C01819=1068.926,-95.070,-58.479,172.290,23.008,154.216
C01820=1068.921,-95.321,-58.468,172.288,23.007,154.216
C01821=1068.914,-95.570,-58.458,172.287,23.005,154.216
C01822=1068.909,-95.820,-58.448,172.285,23.004,154.216
C01823=1068.902,-96.069,-58.438,172.284,23.003,154.216
C01824=1068.897,-96.318,-58.427,172.282,23.001,154.216
C01825=1068.890,-96.568,-58.417,172.280,23.000,154.216
C01826=1068.884,-96.818,-58.406,172.279,22.999,154.216
C01827=1068.878,-97.068,-58.396,172.277,22.997,154.216
C01828=1068.872,-97.318,-58.386,172.275,22.996,154.216
C01829=1068.866,-97.568,-58.376,172.274,22.995,154.216
C01830=1068.859,-97.850,-58.365,172.272,22.993,154.215
C01831=1068.852,-98.133,-58.353,172.270,22.991,154.215
C01832=1068.845,-98.416,-58.341,172.268,22.990,154.215
C01833=1068.838,-98.698,-58.330,172.267,22.989,154.215
C01834=1068.833,-98.948,-58.319,172.265,22.987,154.215
C01835=1068.827,-99.197,-58.309,172.263,22.986,154.215
C01836=1068.820,-99.447,-58.299,172.261,22.985,154.215
C01837=1068.814,-99.697,-58.289,172.260,22.984,154.215
C01838=1068.808,-99.947,-58.278,172.258,22.982,154.215
C01839=1068.801,-100.196,-58.269,172.257,22.981,154.215
C01840=1068.796,-100.446,-58.258,172.255,22.980,154.215
C01841=1068.789,-100.696,-58.248,172.253,22.978,154.215
C01842=1068.783,-100.945,-58.239,172.252,22.977,154.215
C01843=1068.777,-101.195,-58.229,172.250,22.976,154.215
C01844=1068.771,-101.445,-58.218,172.248,22.975,154.215
C01845=1068.764,-101.695,-58.208,172.247,22.974,154.215
C01846=1068.758,-101.944,-58.198,172.245,22.972,154.215
C01847=1068.753,-102.194,-58.188,172.243,22.971,154.215
C01848=1068.746,-102.444,-58.178,172.242,22.970,154.215
C01849=1068.740,-102.693,-58.168,172.240,22.968,154.215
C01850=1068.734,-102.943,-58.157,172.238,22.968,154.216
C01851=1068.728,-103.193,-58.148,172.237,22.966,154.215
C01852=1068.722,-103.443,-58.138,172.235,22.965,154.215
C01853=1068.716,-103.692,-58.127,172.234,22.964,154.215
C01854=1068.710,-103.942,-58.118,172.232,22.962,154.215
C01855=1068.704,-104.192,-58.108,172.230,22.961,154.215
C01856=1068.697,-104.441,-58.098,172.228,22.960,154.216
C01857=1068.692,-104.691,-58.088,172.227,22.959,154.216
C01858=1068.686,-104.941,-58.078,172.225,22.958,154.216
C01859=1068.680,-105.191,-58.069,172.224,22.956,154.216
C01860=1068.673,-105.440,-58.058,172.222,22.956,154.216
C01861=1068.667,-105.691,-58.048,172.220,22.954,154.216
C01862=1068.661,-105.940,-58.038,172.219,22.953,154.216
C01863=1068.654,-106.189,-58.028,172.217,22.952,154.216
C01864=1068.648,-106.439,-58.018,172.215,22.951,154.216
C01865=1068.643,-106.689,-58.008,172.213,22.949,154.216
C01866=1068.637,-106.939,-57.999,172.212,22.948,154.216
C01867=1068.630,-107.188,-57.988,172.210,22.947,154.216
C01868=1068.624,-107.438,-57.979,172.208,22.946,154.216
C01869=1068.618,-107.688,-57.969,172.207,22.945,154.216
C01870=1068.612,-107.938,-57.959,172.205,22.943,154.216
C01871=1068.606,-108.188,-57.949,172.203,22.943,154.216
C01872=1068.600,-108.437,-57.939,172.202,22.941,154.216
C01873=1068.594,-108.687,-57.930,172.200,22.940,154.216
C01874=1068.587,-108.937,-57.920,172.198,22.939,154.216
C01875=1068.581,-109.186,-57.910,172.197,22.938,154.216
C01876=1068.575,-109.436,-57.901,172.195,22.937,154.216
C01877=1068.569,-109.685,-57.891,172.193,22.936,154.216
C01878=1068.562,-109.935,-57.881,172.191,22.935,154.216
C01879=1068.557,-110.185,-57.871,172.190,22.934,154.216
C01880=1068.551,-110.435,-57.861,172.188,22.932,154.216
C01881=1068.545,-110.685,-57.852,172.187,22.932,154.216
C01882=1068.539,-110.935,-57.842,172.186,22.931,154.216
C01883=1068.532,-111.185,-57.833,172.184,22.930,154.216
C01884=1068.526,-111.434,-57.822,172.182,22.929,154.216
C01885=1068.520,-111.683,-57.813,172.181,22.928,154.216
C01886=1068.514,-111.933,-57.803,172.179,22.926,154.216
C01887=1068.507,-112.183,-57.794,172.177,22.925,154.216
C01888=1068.501,-112.433,-57.784,172.175,22.924,154.216
C01889=1068.495,-112.683,-57.774,172.174,22.923,154.216
C01890=1068.490,-112.933,-57.764,172.172,22.922,154.217
C01891=1068.483,-113.183,-57.755,172.170,22.921,154.217
C01892=1068.478,-113.432,-57.746,172.169,22.920,154.217
C01893=1068.472,-113.681,-57.736,172.167,22.919,154.217
C01894=1068.465,-113.962,-57.725,172.165,22.918,154.217
C01895=1068.458,-114.243,-57.714,172.163,22.916,154.217
C01896=1068.450,-114.522,-57.704,172.161,22.916,154.217
C01897=1068.443,-114.803,-57.693,172.159,22.914,154.217
C01898=1068.437,-115.053,-57.683,172.157,22.913,154.217
C01899=1068.431,-115.303,-57.674,172.156,22.912,154.217
C01900=1068.425,-115.552,-57.664,172.154,22.911,154.217
C01901=1068.419,-115.802,-57.654,172.152,22.910,154.217
C01902=1068.413,-116.052,-57.645,172.151,22.909,154.217
C01903=1068.406,-116.302,-57.635,172.149,22.909,154.217
C01904=1068.400,-116.552,-57.626,172.147,22.907,154.217
C01905=1068.395,-116.801,-57.616,172.145,22.906,154.217
C01906=1068.389,-117.050,-57.607,172.144,22.906,154.218
C01907=1068.382,-117.300,-57.597,172.143,22.905,154.217
C01908=1068.376,-117.550,-57.588,172.141,22.904,154.218
C01909=1068.370,-117.800,-57.578,172.139,22.903,154.218
C01910=1068.364,-118.050,-57.569,172.138,22.902,154.218
C01911=1068.358,-118.300,-57.560,172.136,22.901,154.218
C01912=1068.351,-118.550,-57.551,172.134,22.900,154.218
C01913=1068.345,-118.799,-57.541,172.132,22.899,154.218
C01914=1068.339,-119.049,-57.532,172.131,22.898,154.218
C01915=1068.333,-119.298,-57.522,172.129,22.897,154.218
C01916=1068.327,-119.548,-57.513,172.127,22.896,154.218
C01917=1068.321,-119.798,-57.503,172.125,22.895,154.218
C01918=1068.315,-120.048,-57.494,172.124,22.895,154.218
C01919=1068.308,-120.297,-57.484,172.122,22.893,154.218
C01920=1068.303,-120.548,-57.475,172.120,22.893,154.218
C01921=1068.296,-120.798,-57.466,172.118,22.892,154.219
C01922=1068.289,-121.047,-57.457,172.117,22.890,154.219
C01923=1068.284,-121.296,-57.448,172.115,22.890,154.219
C01924=1068.278,-121.546,-57.438,172.113,22.889,154.219
C01925=1068.272,-121.796,-57.428,172.111,22.888,154.219
C01926=1068.265,-122.046,-57.419,172.110,22.887,154.219
C01927=1068.260,-122.296,-57.410,172.109,22.886,154.219
C01928=1068.253,-122.546,-57.401,172.107,22.886,154.219
C01929=1068.247,-122.795,-57.392,172.105,22.885,154.219
C01930=1068.241,-123.044,-57.382,172.103,22.884,154.219
C01931=1068.235,-123.294,-57.373,172.102,22.883,154.219
C01932=1068.229,-123.545,-57.364,172.100,22.882,154.219
C01933=1068.223,-123.794,-57.354,172.098,22.881,154.219
C01934=1068.217,-124.044,-57.345,172.096,22.880,154.220
C01935=1068.210,-124.293,-57.336,172.095,22.880,154.220
C01936=1068.204,-124.543,-57.327,172.093,22.879,154.220
C01937=1068.198,-124.793,-57.318,172.091,22.878,154.220
C01938=1068.192,-125.043,-57.308,172.089,22.877,154.220
C01939=1068.185,-125.292,-57.299,172.088,22.876,154.220
C01940=1068.180,-125.542,-57.291,172.086,22.875,154.220
C01941=1068.174,-125.792,-57.281,172.084,22.875,154.220
C01942=1068.167,-126.042,-57.272,172.083,22.874,154.220
C01943=1068.161,-126.291,-57.263,172.081,22.873,154.220
C01944=1068.155,-126.542,-57.254,172.079,22.873,154.221
C01945=1068.149,-126.791,-57.244,172.078,22.872,154.221
C01946=1068.142,-127.040,-57.236,172.076,22.871,154.221
C01947=1068.136,-127.291,-57.227,172.074,22.870,154.221
C01948=1068.130,-127.540,-57.217,172.072,22.870,154.221
C01949=1068.124,-127.790,-57.208,172.070,22.869,154.221
C01950=1068.118,-128.041,-57.199,172.069,22.868,154.221
C01951=1068.115,-128.291,-57.188,172.067,22.866,154.221
C01952=1068.113,-128.542,-57.178,172.066,22.863,154.221
C01953=1068.113,-128.793,-57.166,172.065,22.860,154.220
C01954=1068.115,-129.046,-57.153,172.064,22.856,154.220
C01955=1068.119,-129.298,-57.140,172.064,22.852,154.219
C01956=1068.125,-129.549,-57.125,172.064,22.847,154.218
C01957=1068.132,-129.799,-57.110,172.064,22.841,154.217
C01958=1067.743,-129.822,-57.282,172.016,22.987,154.250
C01959=1067.737,-129.572,-57.297,172.017,22.993,154.251
C01960=1067.732,-129.320,-57.312,172.017,22.997,154.252
C01961=1067.727,-129.068,-57.325,172.018,23.002,154.252
C01962=1067.725,-128.816,-57.338,172.018,23.005,154.253
C01963=1067.725,-128.565,-57.350,172.019,23.009,154.254
C01964=1067.726,-128.314,-57.361,172.020,23.011,154.254
C01965=1067.730,-128.063,-57.371,172.021,23.013,154.254
C01966=1067.736,-127.812,-57.381,172.023,23.014,154.254
C01967=1067.742,-127.563,-57.390,172.025,23.015,154.254
C01968=1067.747,-127.313,-57.399,172.027,23.015,154.254
C01969=1067.754,-127.063,-57.408,172.029,23.016,154.254
C01970=1067.760,-126.814,-57.417,172.030,23.017,154.253
C01971=1067.766,-126.564,-57.427,172.032,23.018,154.253
C01972=1067.773,-126.314,-57.436,172.034,23.018,154.253
C01973=1067.778,-126.065,-57.444,172.036,23.019,154.253
C01974=1067.785,-125.815,-57.454,172.037,23.021,154.253
C01975=1067.791,-125.565,-57.463,172.039,23.021,154.253
C01976=1067.797,-125.315,-57.472,172.040,23.022,154.253
C01977=1067.804,-125.065,-57.481,172.042,23.022,154.253
C01978=1067.810,-124.815,-57.491,172.044,23.023,154.253
C01979=1067.815,-124.566,-57.500,172.045,23.024,154.253
C01980=1067.822,-124.316,-57.508,172.047,23.025,154.252
C01981=1067.828,-124.066,-57.518,172.049,23.025,154.252
C01982=1067.834,-123.816,-57.527,172.051,23.027,154.252
C01983=1067.840,-123.567,-57.537,172.053,23.028,154.252
C01984=1067.846,-123.317,-57.545,172.054,23.028,154.252
C01985=1067.852,-123.067,-57.555,172.056,23.029,154.252
C01986=1067.859,-122.818,-57.564,172.058,23.030,154.252
C01987=1067.865,-122.568,-57.573,172.060,23.031,154.252
C01988=1067.871,-122.318,-57.583,172.061,23.032,154.252
C01989=1067.877,-122.068,-57.593,172.063,23.033,154.252
C01990=1067.883,-121.819,-57.601,172.065,23.033,154.252
C01991=1067.889,-121.569,-57.611,172.067,23.034,154.251
C01992=1067.896,-121.319,-57.620,172.068,23.035,154.251
C01993=1067.902,-121.069,-57.629,172.070,23.036,154.251
C01994=1067.908,-120.820,-57.639,172.071,23.037,154.251
C01995=1067.914,-120.570,-57.648,172.073,23.038,154.251
C01996=1067.920,-120.319,-57.657,172.075,23.039,154.251
C01997=1067.926,-120.070,-57.666,172.076,23.039,154.251
C01998=1067.932,-119.821,-57.676,172.078,23.040,154.251
C01999=1067.938,-119.571,-57.685,172.080,23.042,154.251
C02000=1067.944,-119.321,-57.695,172.082,23.042,154.251
C02001=1067.951,-119.071,-57.704,172.083,23.043,154.251
C02002=1067.957,-118.822,-57.714,172.085,23.044,154.251
C02003=1067.963,-118.572,-57.723,172.087,23.045,154.251
C02004=1067.970,-118.322,-57.733,172.089,23.046,154.251
C02005=1067.976,-118.072,-57.742,172.090,23.047,154.251
C02006=1067.981,-117.823,-57.751,172.092,23.048,154.250
C02007=1067.987,-117.573,-57.760,172.094,23.049,154.250
C02008=1067.993,-117.323,-57.770,172.095,23.050,154.250
C02009=1067.999,-117.073,-57.779,172.097,23.051,154.250
C02010=1068.006,-116.823,-57.789,172.099,23.052,154.250
C02011=1068.012,-116.574,-57.799,172.101,23.053,154.250
C02012=1068.018,-116.324,-57.808,172.103,23.054,154.250
C02013=1068.024,-116.074,-57.818,172.104,23.055,154.250
C02014=1068.030,-115.824,-57.827,172.106,23.056,154.250
C02015=1068.037,-115.574,-57.837,172.108,23.056,154.250
C02016=1068.043,-115.325,-57.846,172.109,23.058,154.250
C02017=1068.049,-115.075,-57.856,172.110,23.058,154.250
C02018=1068.054,-114.826,-57.865,172.112,23.059,154.250
C02019=1068.062,-114.545,-57.876,172.115,23.061,154.250
C02020=1068.069,-114.265,-57.887,172.116,23.062,154.250
C02021=1068.076,-113.984,-57.898,172.118,23.063,154.249
C02022=1068.083,-113.703,-57.908,172.120,23.064,154.250
C02023=1068.089,-113.453,-57.918,172.122,23.065,154.249
C02024=1068.095,-113.205,-57.928,172.123,23.066,154.249
C02025=1068.101,-112.955,-57.937,172.125,23.067,154.249
C02026=1068.107,-112.705,-57.947,172.127,23.068,154.249
C02027=1068.113,-112.455,-57.957,172.128,23.069,154.249
C02028=1068.119,-112.205,-57.967,172.130,23.070,154.249
C02029=1068.125,-111.955,-57.976,172.132,23.072,154.249
C02030=1068.131,-111.706,-57.986,172.133,23.072,154.249
C02031=1068.137,-111.456,-57.995,172.135,23.074,154.249
C02032=1068.144,-111.206,-58.005,172.137,23.074,154.249
C02033=1068.150,-110.956,-58.014,172.139,23.076,154.249
C02034=1068.156,-110.707,-58.025,172.140,23.076,154.249
C02035=1068.162,-110.457,-58.034,172.142,23.078,154.249
C02036=1068.169,-110.207,-58.044,172.144,23.079,154.249
C02037=1068.175,-109.958,-58.053,172.145,23.080,154.249
C02038=1068.180,-109.707,-58.063,172.147,23.081,154.249
C02039=1068.186,-109.458,-58.073,172.149,23.082,154.249
C02040=1068.193,-109.208,-58.083,172.150,23.083,154.249
C02041=1068.199,-108.959,-58.093,172.152,23.085,154.249
C02042=1068.205,-108.709,-58.102,172.154,23.085,154.249
C02043=1068.211,-108.459,-58.112,172.155,23.087,154.249
C02044=1068.218,-108.209,-58.122,172.157,23.087,154.249
C02045=1068.224,-107.960,-58.132,172.159,23.089,154.249
C02046=1068.229,-107.710,-58.142,172.161,23.090,154.249
C02047=1068.236,-107.460,-58.152,172.162,23.091,154.248
C02048=1068.242,-107.210,-58.161,172.164,23.092,154.248
C02049=1068.248,-106.961,-58.171,172.166,23.093,154.248
C02050=1068.254,-106.711,-58.181,172.167,23.094,154.248
C02051=1068.260,-106.461,-58.191,172.169,23.096,154.248
C02052=1068.266,-106.212,-58.201,172.171,23.097,154.248
C02053=1068.273,-105.962,-58.211,172.172,23.098,154.248
C02054=1068.279,-105.713,-58.221,172.174,23.099,154.248
C02055=1068.285,-105.462,-58.231,172.176,23.100,154.248
C02056=1068.291,-105.212,-58.241,172.177,23.102,154.248
C02057=1068.297,-104.963,-58.251,172.179,23.103,154.248
C02058=1068.304,-104.713,-58.261,172.181,23.104,154.248
C02059=1068.309,-104.463,-58.271,172.182,23.105,154.248
C02060=1068.315,-104.214,-58.281,172.184,23.106,154.248
C02061=1068.322,-103.964,-58.291,172.185,23.107,154.248
C02062=1068.328,-103.714,-58.300,172.186,23.109,154.248
C02063=1068.334,-103.465,-58.311,172.188,23.109,154.248
C02064=1068.340,-103.215,-58.321,172.190,23.111,154.248
C02065=1068.346,-102.965,-58.330,172.192,23.112,154.248
C02066=1068.352,-102.715,-58.341,172.193,23.113,154.248
C02067=1068.358,-102.466,-58.351,172.195,23.115,154.248
C02068=1068.364,-102.216,-58.360,172.196,23.116,154.248
C02069=1068.370,-101.967,-58.370,172.198,23.117,154.248
C02070=1068.376,-101.717,-58.381,172.200,23.118,154.248
C02071=1068.383,-101.467,-58.391,172.201,23.119,154.248
C02072=1068.389,-101.217,-58.401,172.203,23.121,154.248
C02073=1068.395,-100.967,-58.411,172.205,23.122,154.248
C02074=1068.401,-100.718,-58.421,172.206,23.123,154.248
C02075=1068.407,-100.468,-58.431,172.208,23.125,154.248
C02076=1068.413,-100.218,-58.442,172.210,23.126,154.248
C02077=1068.419,-99.969,-58.451,172.211,23.127,154.248
C02078=1068.426,-99.719,-58.462,172.213,23.128,154.248
C02079=1068.432,-99.469,-58.472,172.215,23.129,154.248
C02080=1068.438,-99.219,-58.482,172.216,23.131,154.248
C02081=1068.444,-98.970,-58.492,172.218,23.132,154.248
C02082=1068.450,-98.719,-58.502,172.220,23.133,154.248
C02083=1068.457,-98.436,-58.514,172.222,23.135,154.248
C02084=1068.464,-98.154,-58.525,172.224,23.136,154.248
C02085=1068.471,-97.871,-58.537,172.225,23.138,154.248
C02086=1068.477,-97.589,-58.548,172.227,23.139,154.248
C02087=1068.484,-97.339,-58.559,172.230,23.141,154.248
C02088=1068.490,-97.089,-58.569,172.231,23.142,154.248
C02089=1068.496,-96.840,-58.579,172.233,23.143,154.248
C02090=1068.502,-96.590,-58.590,172.234,23.145,154.248
C02091=1068.508,-96.341,-58.600,172.236,23.147,154.248
C02092=1068.514,-96.091,-58.611,172.238,23.148,154.248
C02093=1068.520,-95.841,-58.620,172.239,23.149,154.248
C02094=1068.526,-95.592,-58.631,172.241,23.150,154.248
C02095=1068.532,-95.341,-58.641,172.242,23.152,154.248
C02096=1068.538,-95.092,-58.652,172.244,23.153,154.249
C02097=1068.544,-94.842,-58.663,172.246,23.154,154.249
C02098=1068.550,-94.592,-58.672,172.247,23.156,154.249
C02099=1068.556,-94.343,-58.683,172.249,23.157,154.249
C02100=1068.562,-94.093,-58.693,172.250,23.159,154.249
C02101=1068.568,-93.844,-58.704,172.252,23.160,154.249
C02102=1068.575,-93.594,-58.714,172.254,23.162,154.249
C02103=1068.580,-93.344,-58.724,172.255,23.163,154.249
C02104=1068.586,-93.094,-58.735,172.257,23.164,154.249
C02105=1068.592,-92.844,-58.745,172.259,23.166,154.249
C02106=1068.598,-92.595,-58.756,172.260,23.167,154.249
C02107=1068.605,-92.345,-58.766,172.262,23.169,154.249
C02108=1068.611,-92.095,-58.776,172.263,23.170,154.249
C02109=1068.616,-91.845,-58.787,172.265,23.171,154.249
C02110=1068.623,-91.596,-58.798,172.267,23.173,154.249
C02111=1068.629,-91.347,-58.809,172.268,23.174,154.249
C02112=1068.635,-91.096,-58.818,172.270,23.176,154.249
C02113=1068.641,-90.847,-58.829,172.271,23.177,154.249
C02114=1068.647,-90.597,-58.840,172.273,23.179,154.249
C02115=1068.653,-90.347,-58.850,172.275,23.180,154.249
C02116=1068.659,-90.098,-58.861,172.276,23.181,154.249
C02117=1068.666,-89.848,-58.871,172.278,23.183,154.249
C02118=1068.671,-89.599,-58.882,172.279,23.184,154.249
C02119=1068.677,-89.349,-58.892,172.281,23.186,154.249
C02120=1068.683,-89.099,-58.903,172.283,23.187,154.249
C02121=1068.690,-88.849,-58.914,172.284,23.189,154.250
C02122=1068.696,-88.600,-58.924,172.286,23.190,154.250
C02123=1068.702,-88.350,-58.934,172.287,23.192,154.250
C02124=1068.707,-88.100,-58.945,172.289,23.193,154.250
C02125=1068.714,-87.850,-58.956,172.290,23.195,154.250
C02126=1068.720,-87.601,-58.967,172.292,23.196,154.250
C02127=1068.726,-87.352,-58.978,172.294,23.197,154.250
C02128=1068.733,-87.101,-58.988,172.295,23.199,154.250
C02129=1068.738,-86.852,-58.998,172.297,23.201,154.250
C02130=1068.744,-86.602,-59.009,172.298,23.202,154.250
C02131=1068.751,-86.353,-59.020,172.300,23.203,154.250
C02132=1068.757,-86.103,-59.031,172.301,23.205,154.250
C02133=1068.762,-85.853,-59.041,172.303,23.206,154.250
C02134=1068.769,-85.603,-59.051,172.305,23.208,154.250
C02135=1068.775,-85.353,-59.062,172.306,23.209,154.250
C02136=1068.781,-85.104,-59.073,172.308,23.211,154.250
C02137=1068.787,-84.855,-59.084,172.309,23.212,154.250
C02138=1068.794,-84.604,-59.095,172.311,23.214,154.250
C02139=1068.800,-84.355,-59.106,172.313,23.215,154.250
C02140=1068.806,-84.106,-59.116,172.314,23.217,154.250
C02141=1068.812,-83.855,-59.127,172.316,23.218,154.251
C02142=1068.818,-83.605,-59.137,172.317,23.220,154.251
C02143=1068.824,-83.356,-59.148,172.320,23.222,154.251
C02144=1068.831,-83.106,-59.159,172.321,23.223,154.251
C02145=1068.836,-82.856,-59.170,172.323,23.225,154.251
C02146=1068.843,-82.607,-59.180,172.325,23.226,154.251
C02147=1068.850,-82.326,-59.193,172.326,23.228,154.251
C02148=1068.857,-82.046,-59.205,172.328,23.229,154.251
C02149=1068.864,-81.766,-59.217,172.329,23.231,154.251
C02150=1068.871,-81.486,-59.229,172.332,23.233,154.251
C02151=1068.877,-81.235,-59.241,172.333,23.235,154.251
C02152=1068.883,-80.986,-59.251,172.335,23.236,154.251
C02153=1068.889,-80.737,-59.262,172.336,23.238,154.251
C02154=1068.895,-80.487,-59.273,172.338,23.239,154.251
C02155=1068.902,-80.237,-59.283,172.339,23.241,154.251
C02156=1068.908,-79.987,-59.295,172.341,23.243,154.252
C02157=1068.914,-79.738,-59.306,172.343,23.244,154.252
C02158=1068.920,-79.488,-59.316,172.344,23.246,154.252
C02159=1068.926,-79.238,-59.328,172.346,23.247,154.252
C02160=1068.932,-78.989,-59.339,172.347,23.249,154.252
C02161=1068.938,-78.739,-59.349,172.349,23.250,154.252
C02162=1068.945,-78.489,-59.360,172.350,23.252,154.252
C02163=1068.950,-78.240,-59.371,172.352,23.254,154.252
C02164=1068.957,-77.990,-59.382,172.353,23.255,154.252
C02165=1068.962,-77.740,-59.393,172.355,23.257,154.252
C02166=1068.968,-77.491,-59.404,172.356,23.259,154.252
C02167=1068.975,-77.240,-59.415,172.358,23.260,154.253
C02168=1068.980,-76.991,-59.426,172.360,23.262,154.253
C02169=1068.986,-76.741,-59.437,172.361,23.264,154.253
C02170=1068.993,-76.492,-59.449,172.363,23.266,154.253
C02171=1068.998,-76.242,-59.460,172.365,23.267,154.253
C02172=1069.005,-75.992,-59.471,172.366,23.269,154.253
C02173=1069.010,-75.743,-59.482,172.368,23.270,154.253
C02174=1069.017,-75.492,-59.493,172.370,23.272,154.253
C02175=1069.023,-75.243,-59.503,172.371,23.274,154.253
C02176=1069.029,-74.994,-59.514,172.373,23.275,154.253
C02177=1069.036,-74.744,-59.526,172.374,23.277,154.253
C02178=1069.041,-74.495,-59.537,172.376,23.279,154.253
C02179=1069.048,-74.245,-59.548,172.377,23.281,154.254
C02180=1069.054,-73.995,-59.559,172.379,23.282,154.254
C02181=1069.060,-73.745,-59.570,172.380,23.284,154.254
C02182=1069.066,-73.496,-59.582,172.382,23.286,154.254
C02183=1069.071,-73.246,-59.594,172.383,23.287,154.254
C02184=1069.077,-72.996,-59.605,172.385,23.289,154.254
C02185=1069.083,-72.747,-59.616,172.386,23.291,154.254
C02186=1069.089,-72.496,-59.627,172.388,23.293,154.254
C02187=1069.095,-72.247,-59.638,172.389,23.294,154.254
C02188=1069.101,-71.998,-59.649,172.391,23.296,154.255
C02189=1069.107,-71.747,-59.661,172.392,23.298,154.255
C02190=1069.112,-71.498,-59.672,172.394,23.299,154.255
C02191=1069.119,-71.248,-59.684,172.395,23.301,154.255
C02192=1069.125,-70.999,-59.695,172.397,23.303,154.255
C02193=1069.131,-70.749,-59.706,172.399,23.305,154.255
C02194=1069.137,-70.500,-59.718,172.401,23.307,154.255
C02195=1069.142,-70.250,-59.729,172.402,23.309,154.255
C02196=1069.149,-70.000,-59.740,172.404,23.311,154.255
C02197=1069.155,-69.751,-59.752,172.405,23.312,154.256
C02198=1069.161,-69.501,-59.763,172.407,23.314,154.256
C02199=1069.167,-69.251,-59.774,172.408,23.316,154.256
C02200=1069.173,-69.002,-59.786,172.410,23.318,154.256
C02201=1069.178,-68.752,-59.798,172.411,23.320,154.256
C02202=1069.185,-68.502,-59.809,172.413,23.321,154.256
C02203=1069.191,-68.253,-59.820,172.414,23.323,154.256
C02204=1069.197,-68.003,-59.832,172.416,23.325,154.256
C02205=1069.203,-67.753,-59.843,172.417,23.327,154.257
C02206=1069.209,-67.503,-59.855,172.419,23.329,154.257
C02207=1069.214,-67.254,-59.866,172.420,23.331,154.257
C02208=1069.221,-67.004,-59.878,172.421,23.333,154.257
C02209=1069.227,-66.755,-59.889,172.423,23.334,154.257
C02210=1069.232,-66.504,-59.901,172.425,23.336,154.257
C02211=1069.239,-66.227,-59.913,172.427,23.339,154.257
C02212=1069.246,-65.949,-59.927,172.428,23.340,154.258
C02213=1069.253,-65.670,-59.939,172.430,23.342,154.258
C02214=1069.259,-65.392,-59.952,172.432,23.345,154.258
C02215=1069.265,-65.142,-59.963,172.434,23.346,154.258
C02216=1069.272,-64.893,-59.975,172.435,23.348,154.258
C02217=1069.278,-64.643,-59.986,172.436,23.350,154.258
C02218=1069.283,-64.393,-59.998,172.438,23.352,154.258
C02219=1069.289,-64.144,-60.009,172.440,23.353,154.258
C02220=1069.296,-63.894,-60.021,172.441,23.355,154.259
C02221=1069.302,-63.645,-60.032,172.443,23.357,154.259
C02222=1069.307,-63.395,-60.045,172.444,23.359,154.259
C02223=1069.314,-63.145,-60.056,172.445,23.361,154.259
C02224=1069.320,-62.896,-60.068,172.447,23.363,154.259
C02225=1069.326,-62.645,-60.079,172.448,23.365,154.259
C02226=1069.332,-62.396,-60.091,172.450,23.366,154.259
C02227=1069.338,-62.146,-60.102,172.451,23.368,154.260
C02228=1069.345,-61.897,-60.114,172.453,23.370,154.260
C02229=1069.350,-61.647,-60.126,172.454,23.372,154.260
C02230=1069.356,-61.397,-60.138,172.456,23.374,154.260
C02231=1069.362,-61.148,-60.149,172.458,23.376,154.260
C02232=1069.369,-60.898,-60.160,172.460,23.378,154.260
C02233=1069.374,-60.648,-60.173,172.461,23.380,154.260
C02234=1069.380,-60.399,-60.184,172.463,23.382,154.261
C02235=1069.387,-60.149,-60.196,172.464,23.384,154.261
C02236=1069.392,-59.900,-60.208,172.465,23.386,154.261
C02237=1069.398,-59.650,-60.219,172.467,23.387,154.261
C02238=1069.405,-59.400,-60.231,172.468,23.389,154.261
C02239=1069.411,-59.151,-60.242,172.470,23.391,154.261
C02240=1069.417,-58.901,-60.255,172.471,23.393,154.261
C02241=1069.423,-58.651,-60.267,172.473,23.395,154.262
C02242=1069.429,-58.402,-60.278,172.474,23.397,154.262
C02243=1069.435,-58.152,-60.290,172.476,23.399,154.262
C02244=1069.442,-57.902,-60.302,172.477,23.400,154.262
C02245=1069.447,-57.653,-60.313,172.479,23.402,154.262
C02246=1069.453,-57.403,-60.325,172.480,23.404,154.262
C02247=1069.460,-57.153,-60.337,172.482,23.406,154.263
C02248=1069.466,-56.904,-60.348,172.484,23.408,154.263
C02249=1069.472,-56.654,-60.361,172.485,23.410,154.263
C02250=1069.478,-56.404,-60.373,172.487,23.412,154.263
C02251=1069.485,-56.155,-60.385,172.488,23.414,154.263
C02252=1069.490,-55.905,-60.396,172.490,23.416,154.263
C02253=1069.497,-55.655,-60.408,172.491,23.418,154.263
C02254=1069.503,-55.406,-60.420,172.493,23.420,154.263
C02255=1069.509,-55.157,-60.432,172.494,23.421,154.264
C02256=1069.515,-54.907,-60.444,172.496,23.423,154.264
C02257=1069.522,-54.657,-60.456,172.497,23.425,154.264
C02258=1069.527,-54.407,-60.468,172.499,23.428,154.264
C02259=1069.534,-54.158,-60.480,172.500,23.429,154.264
C02260=1069.540,-53.908,-60.491,172.502,23.431,154.264
C02261=1069.546,-53.658,-60.504,172.503,23.433,154.265
C02262=1069.552,-53.409,-60.515,172.504,23.435,154.265
C02263=1069.558,-53.160,-60.527,172.507,23.437,154.265
C02264=1069.564,-52.910,-60.540,172.508,23.439,154.265
C02265=1069.571,-52.660,-60.551,172.510,23.441,154.265
C02266=1069.577,-52.410,-60.563,172.511,23.443,154.265
C02267=1069.583,-52.161,-60.575,172.513,23.445,154.265
C02268=1069.589,-51.911,-60.587,172.514,23.447,154.266
C02269=1069.595,-51.661,-60.600,172.516,23.449,154.266
C02270=1069.602,-51.412,-60.611,172.517,23.451,154.266
C02271=1069.608,-51.162,-60.624,172.518,23.453,154.266
C02272=1069.613,-50.912,-60.635,172.520,23.455,154.266
C02273=1069.620,-50.663,-60.647,172.521,23.457,154.266
C02274=1069.626,-50.413,-60.659,172.523,23.458,154.267
C02275=1069.633,-50.136,-60.673,172.525,23.461,154.267
C02276=1069.639,-49.859,-60.686,172.527,23.463,154.267
C02277=1069.646,-49.583,-60.700,172.528,23.466,154.267
C02278=1069.653,-49.306,-60.713,172.529,23.467,154.267
C02279=1069.659,-49.056,-60.726,172.532,23.470,154.268
C02280=1069.665,-48.806,-60.738,172.533,23.472,154.268
C02281=1069.671,-48.557,-60.750,172.534,23.474,154.268
C02282=1069.677,-48.307,-60.763,172.536,23.476,154.268
C02283=1069.683,-48.058,-60.775,172.537,23.478,154.268
C02284=1069.689,-47.808,-60.787,172.539,23.480,154.269
C02285=1069.694,-47.558,-60.799,172.540,23.483,154.269
C02286=1069.701,-47.309,-60.811,172.542,23.484,154.269
C02287=1069.707,-47.059,-60.824,172.543,23.486,154.269
C02288=1069.713,-46.809,-60.836,172.544,23.489,154.269
C02289=1069.719,-46.560,-60.848,172.546,23.491,154.270
C02290=1069.725,-46.310,-60.861,172.547,23.492,154.270
C02291=1069.731,-46.060,-60.873,172.549,23.495,154.270
C02292=1069.737,-45.811,-60.885,172.550,23.497,154.270
C02293=1069.743,-45.561,-60.898,172.552,23.499,154.270
C02294=1069.749,-45.312,-60.910,172.554,23.501,154.270
C02295=1069.755,-45.062,-60.922,172.555,23.503,154.271
C02296=1069.761,-44.812,-60.934,172.557,23.505,154.271
C02297=1069.767,-44.562,-60.947,172.558,23.508,154.271
C02298=1069.773,-44.313,-60.959,172.559,23.509,154.271
C02299=1069.779,-44.064,-60.971,172.561,23.512,154.271
C02300=1069.785,-43.814,-60.984,172.562,23.514,154.272
C02301=1069.791,-43.564,-60.996,172.564,23.516,154.272
C02302=1069.797,-43.314,-61.009,172.565,23.518,154.272
C02303=1069.803,-43.065,-61.021,172.567,23.520,154.272
C02304=1069.810,-42.815,-61.034,172.568,23.522,154.272
C02305=1069.815,-42.566,-61.046,172.569,23.524,154.273
C02306=1069.821,-42.316,-61.059,172.571,23.526,154.273
C02307=1069.827,-42.067,-61.071,172.572,23.528,154.273
C02308=1069.833,-41.817,-61.083,172.574,23.531,154.273
C02309=1069.839,-41.567,-61.096,172.576,23.533,154.273
C02310=1069.846,-41.317,-61.108,172.577,23.535,154.274
C02311=1069.852,-41.068,-61.121,172.579,23.537,154.274
C02312=1069.858,-40.818,-61.134,172.580,23.539,154.274
C02313=1069.863,-40.569,-61.146,172.582,23.541,154.274
C02314=1069.870,-40.319,-61.158,172.583,23.543,154.274
C02315=1069.876,-40.069,-61.170,172.584,23.545,154.275
C02316=1069.882,-39.820,-61.184,172.586,23.547,154.275
C02317=1069.888,-39.570,-61.196,172.587,23.550,154.275
C02318=1069.894,-39.320,-61.209,172.589,23.552,154.275
C02319=1069.901,-39.071,-61.221,172.590,23.554,154.275
C02320=1069.907,-38.821,-61.233,172.591,23.556,154.276
C02321=1069.913,-38.572,-61.246,172.593,23.558,154.276
C02322=1069.919,-38.322,-61.259,172.595,23.560,154.276
C02323=1069.924,-38.073,-61.271,172.596,23.563,154.276
C02324=1069.930,-37.823,-61.284,172.598,23.565,154.276
C02325=1069.936,-37.574,-61.297,172.599,23.567,154.277
C02326=1069.942,-37.324,-61.310,172.601,23.569,154.277
C02327=1069.948,-37.074,-61.322,172.602,23.571,154.277
C02328=1069.954,-36.825,-61.335,172.603,23.573,154.277
C02329=1069.961,-36.575,-61.347,172.605,23.576,154.277
C02330=1069.967,-36.325,-61.360,172.606,23.578,154.278
C02331=1069.973,-36.076,-61.373,172.608,23.580,154.278
C02332=1069.978,-35.827,-61.385,172.609,23.582,154.278
C02333=1069.984,-35.577,-61.398,172.610,23.584,154.278
C02334=1069.990,-35.327,-61.411,172.612,23.587,154.279
C02335=1069.996,-35.078,-61.424,172.613,23.589,154.279
C02336=1070.002,-34.828,-61.436,172.615,23.591,154.279
C02337=1070.008,-34.578,-61.450,172.617,23.594,154.279
C02338=1070.014,-34.329,-61.462,172.618,23.596,154.279
C02339=1070.021,-34.052,-61.477,172.619,23.598,154.280
C02340=1070.027,-33.775,-61.490,172.621,23.601,154.280
C02341=1070.034,-33.499,-61.505,172.623,23.603,154.280
C02342=1070.040,-33.222,-61.519,172.624,23.606,154.280
C02343=1070.046,-32.973,-61.532,172.626,23.608,154.281
C02344=1070.053,-32.723,-61.545,172.627,23.610,154.281
C02345=1070.058,-32.473,-61.558,172.629,23.612,154.281
C02346=1070.064,-32.223,-61.570,172.630,23.614,154.281
C02347=1070.071,-31.974,-61.584,172.631,23.617,154.282
C02348=1070.076,-31.724,-61.596,172.633,23.619,154.282
C02349=1070.083,-31.475,-61.609,172.634,23.621,154.282
C02350=1070.089,-31.225,-61.622,172.635,23.623,154.282
C02351=1070.095,-30.976,-61.635,172.638,23.626,154.282
C02352=1070.101,-30.726,-61.648,172.639,23.628,154.283
C02353=1070.107,-30.477,-61.661,172.641,23.630,154.283
C02354=1070.113,-30.227,-61.674,172.642,23.632,154.283
C02355=1070.119,-29.978,-61.687,172.643,23.635,154.283
C02356=1070.125,-29.728,-61.699,172.645,23.637,154.283
C02357=1070.131,-29.479,-61.713,172.646,23.639,154.284
C02358=1070.137,-29.229,-61.725,172.647,23.641,154.284
C02359=1070.143,-28.979,-61.739,172.649,23.643,154.284
C02360=1070.149,-28.729,-61.751,172.650,23.646,154.284
C02361=1070.155,-28.480,-61.764,172.652,23.648,154.285
C02362=1070.161,-28.230,-61.777,172.653,23.650,154.285
C02363=1070.168,-27.981,-61.790,172.654,23.652,154.285
C02364=1070.174,-27.732,-61.803,172.657,23.655,154.285
C02365=1070.180,-27.482,-61.816,172.658,23.657,154.286
C02366=1070.186,-27.232,-61.830,172.659,23.659,154.286
C02367=1070.192,-26.982,-61.842,172.661,23.661,154.286
C02368=1070.198,-26.732,-61.856,172.662,23.664,154.286
C02369=1070.204,-26.483,-61.869,172.663,23.666,154.287
C02370=1070.210,-26.233,-61.882,172.665,23.669,154.287
C02371=1070.216,-25.984,-61.895,172.666,23.670,154.287
C02372=1070.221,-25.734,-61.908,172.668,23.673,154.287
C02373=1070.228,-25.485,-61.922,172.669,23.675,154.287
C02374=1070.234,-25.235,-61.935,172.670,23.678,154.288
C02375=1070.240,-24.985,-61.947,172.672,23.680,154.288
C02376=1070.245,-24.736,-61.961,172.673,23.682,154.288
C02377=1070.251,-24.487,-61.975,172.675,23.685,154.288
C02378=1070.257,-24.237,-61.987,172.677,23.687,154.289
C02379=1070.264,-23.987,-62.000,172.678,23.690,154.289
C02380=1070.269,-23.738,-62.014,172.679,23.691,154.289
C02381=1070.275,-23.489,-62.027,172.681,23.694,154.289
C02382=1070.281,-23.239,-62.040,172.682,23.696,154.290
C02383=1070.287,-22.989,-62.054,172.683,23.699,154.290
C02384=1070.293,-22.740,-62.067,172.685,23.701,154.290
C02385=1070.299,-22.489,-62.080,172.686,23.703,154.290
C02386=1070.306,-22.240,-62.093,172.687,23.705,154.291
C02387=1070.311,-21.990,-62.107,172.689,23.708,154.291
C02388=1070.317,-21.741,-62.121,172.690,23.710,154.291
C02389=1070.323,-21.491,-62.133,172.691,23.713,154.291
C02390=1070.329,-21.242,-62.147,172.694,23.715,154.292
C02391=1070.335,-20.993,-62.160,172.695,23.717,154.292
C02392=1070.341,-20.743,-62.173,172.696,23.720,154.292
C02393=1070.347,-20.494,-62.187,172.698,23.722,154.292
C02394=1070.353,-20.243,-62.200,172.699,23.724,154.293
C02395=1070.359,-19.994,-62.214,172.700,23.727,154.293
C02396=1070.365,-19.745,-62.227,172.702,23.729,154.293
C02397=1070.371,-19.495,-62.241,172.703,23.731,154.293
C02398=1070.377,-19.246,-62.254,172.705,23.733,154.294
C02399=1070.383,-18.996,-62.267,172.706,23.736,154.294
C02400=1070.389,-18.746,-62.280,172.707,23.738,154.294
C02401=1070.395,-18.496,-62.294,172.709,23.741,154.295
C02402=1070.402,-18.247,-62.307,172.710,23.743,154.295
C02403=1070.408,-17.970,-62.323,172.712,23.745,154.295
C02404=1070.415,-17.693,-62.338,172.713,23.748,154.295
C02405=1070.421,-17.415,-62.352,172.715,23.751,154.296
C02406=1070.428,-17.138,-62.367,172.717,23.754,154.296
C02407=1070.434,-16.888,-62.381,172.718,23.756,154.296
C02408=1070.440,-16.639,-62.394,172.720,23.758,154.296
C02409=1070.447,-16.389,-62.408,172.721,23.760,154.297
C02410=1070.452,-16.140,-62.422,172.722,23.763,154.297
C02411=1070.458,-15.890,-62.435,172.724,23.765,154.297
C02412=1070.465,-15.641,-62.448,172.725,23.767,154.297
C02413=1070.471,-15.391,-62.462,172.726,23.770,154.298
C02414=1070.476,-15.141,-62.475,172.728,23.772,154.298
C02415=1070.482,-14.891,-62.489,172.729,23.775,154.298
C02416=1070.488,-14.642,-62.502,172.730,23.777,154.298
C02417=1070.494,-14.392,-62.516,172.732,23.779,154.299
C02418=1070.500,-14.143,-62.529,172.734,23.782,154.299
C02419=1070.506,-13.893,-62.543,172.735,23.784,154.299
C02420=1070.512,-13.644,-62.557,172.737,23.786,154.299
C02421=1070.518,-13.394,-62.570,172.738,23.789,154.300
C02422=1070.523,-13.145,-62.584,172.739,23.791,154.300
C02423=1070.530,-12.895,-62.598,172.741,23.794,154.300
C02424=1070.535,-12.645,-62.612,172.742,23.796,154.301
C02425=1070.542,-12.396,-62.625,172.743,23.799,154.301
C02426=1070.547,-12.147,-62.640,172.745,23.801,154.301
C02427=1070.554,-11.897,-62.653,172.746,23.803,154.301
C02428=1070.560,-11.647,-62.667,172.747,23.806,154.302
C02429=1070.566,-11.398,-62.680,172.749,23.808,154.302
C02430=1070.571,-11.149,-62.694,172.750,23.811,154.302
C02431=1070.577,-10.899,-62.708,172.752,23.813,154.302
C02432=1070.584,-10.649,-62.722,172.754,23.816,154.303
C02433=1070.589,-10.399,-62.736,172.755,23.818,154.303
C02434=1070.595,-10.150,-62.749,172.756,23.821,154.303
C02435=1070.601,-9.901,-62.763,172.758,23.823,154.304
C02436=1070.607,-9.650,-62.777,172.759,23.825,154.304
C02437=1070.613,-9.402,-62.791,172.760,23.828,154.304
C02438=1070.619,-9.152,-62.805,172.762,23.830,154.304
C02439=1070.625,-8.903,-62.818,172.763,23.833,154.305
C02440=1070.631,-8.653,-62.832,172.764,23.835,154.305
C02441=1070.637,-8.403,-62.846,172.766,23.837,154.305
C02442=1070.643,-8.154,-62.860,172.767,23.840,154.305
C02443=1070.649,-7.904,-62.874,172.768,23.842,154.306
C02444=1070.655,-7.655,-62.888,172.771,23.845,154.306
C02445=1070.661,-7.405,-62.902,172.772,23.847,154.306
C02446=1070.667,-7.155,-62.916,172.773,23.850,154.307
C02447=1070.673,-6.906,-62.929,172.775,23.852,154.307
C02448=1070.679,-6.657,-62.944,172.776,23.855,154.307
C02449=1070.685,-6.407,-62.957,172.777,23.857,154.307
C02450=1070.691,-6.157,-62.971,172.779,23.859,154.308
C02451=1070.697,-5.908,-62.985,172.780,23.862,154.308
C02452=1070.703,-5.659,-62.999,172.781,23.864,154.308
C02453=1070.709,-5.409,-63.013,172.783,23.867,154.308
C02454=1070.715,-5.159,-63.027,172.784,23.869,154.309
C02455=1070.721,-4.910,-63.040,172.785,23.871,154.309
C02456=1070.727,-4.660,-63.055,172.787,23.874,154.309
C02457=1070.733,-4.411,-63.069,172.789,23.877,154.310
C02458=1070.740,-4.161,-63.083,172.790,23.879,154.310
C02459=1070.745,-3.911,-63.097,172.791,23.881,154.310
C02460=1070.751,-3.662,-63.111,172.793,23.884,154.310
C02461=1070.758,-3.412,-63.125,172.794,23.886,154.311
C02462=1070.763,-3.163,-63.139,172.795,23.889,154.311
C02463=1070.769,-2.914,-63.153,172.797,23.891,154.311
C02464=1070.775,-2.663,-63.168,172.798,23.893,154.311
C02465=1070.781,-2.414,-63.181,172.799,23.896,154.312
C02466=1070.787,-2.165,-63.195,172.801,23.899,154.312
C02467=1070.793,-1.886,-63.211,172.803,23.901,154.312
C02468=1070.800,-1.606,-63.227,172.804,23.904,154.313
C02469=1070.806,-1.328,-63.244,172.805,23.907,154.313
C02470=1070.813,-1.049,-63.259,172.807,23.910,154.313
C02471=1070.819,-0.799,-63.274,172.809,23.913,154.314
C02472=1070.825,-0.550,-63.288,172.810,23.915,154.314
C02473=1070.830,-0.300,-63.301,172.811,23.917,154.314
C02474=1070.837,-0.051,-63.316,172.813,23.920,154.315
C02475=1070.842,0.199,-63.330,172.814,23.923,154.315
C02476=1070.848,0.448,-63.345,172.815,23.925,154.315
C02477=1070.854,0.698,-63.359,172.817,23.928,154.316
C02478=1070.860,0.947,-63.374,172.818,23.930,154.316
C02479=1070.867,1.197,-63.387,172.819,23.932,154.316
C02480=1070.872,1.447,-63.401,172.821,23.935,154.316
C02481=1070.878,1.696,-63.416,172.822,23.938,154.317
C02482=1070.884,1.946,-63.430,172.823,23.940,154.317
C02483=1070.890,2.195,-63.445,172.825,23.942,154.317
C02484=1070.895,2.444,-63.458,172.827,23.945,154.318
C02485=1070.902,2.694,-63.473,172.828,23.948,154.318
C02486=1070.907,2.944,-63.487,172.829,23.951,154.318
C02487=1070.913,3.193,-63.502,172.831,23.953,154.319
C02488=1070.919,3.442,-63.517,172.832,23.955,154.319
C02489=1070.925,3.692,-63.531,172.833,23.958,154.319
C02490=1070.931,3.941,-63.546,172.835,23.960,154.319
C02491=1070.937,4.191,-63.559,172.836,23.963,154.320
C02492=1070.943,4.441,-63.574,172.837,23.965,154.320
C02493=1070.948,4.690,-63.588,172.839,23.968,154.320
C02494=1070.955,4.940,-63.603,172.840,23.970,154.321
C02495=1070.960,5.190,-63.617,172.841,23.973,154.321
C02496=1070.967,5.439,-63.632,172.843,23.975,154.321
C02497=1070.972,5.688,-63.647,172.845,23.978,154.321
C02498=1070.978,5.938,-63.660,172.846,23.981,154.322
C02499=1070.984,6.187,-63.675,172.847,23.983,154.322
C02500=1070.990,6.437,-63.689,172.849,23.986,154.322
C02501=1070.996,6.687,-63.704,172.850,23.988,154.323
C02502=1071.002,6.936,-63.719,172.851,23.990,154.323
C02503=1071.008,7.186,-63.733,172.853,23.993,154.323
C02504=1071.014,7.435,-63.748,172.854,23.996,154.324
C02505=1071.020,7.684,-63.763,172.855,23.998,154.324
C02506=1071.026,7.934,-63.776,172.857,24.000,154.324
C02507=1071.032,8.184,-63.791,172.858,24.003,154.324
C02508=1071.038,8.433,-63.806,172.859,24.005,154.325
C02509=1071.044,8.683,-63.820,172.860,24.008,154.325
C02510=1071.050,8.932,-63.835,172.863,24.011,154.325
C02511=1071.056,9.181,-63.850,172.864,24.013,154.326
C02512=1071.062,9.430,-63.864,172.865,24.016,154.326
C02513=1071.068,9.681,-63.879,172.867,24.018,154.326
C02514=1071.074,9.930,-63.893,172.868,24.021,154.326
C02515=1071.080,10.179,-63.908,172.869,24.024,154.327
C02516=1071.086,10.429,-63.922,172.871,24.026,154.327
C02517=1071.092,10.679,-63.937,172.872,24.028,154.327
C02518=1071.098,10.928,-63.952,172.873,24.031,154.328
C02519=1071.104,11.177,-63.966,172.875,24.033,154.328
C02520=1071.110,11.427,-63.981,172.876,24.035,154.328
C02521=1071.116,11.676,-63.995,172.877,24.038,154.329
C02522=1071.122,11.926,-64.010,172.879,24.041,154.329
C02523=1071.128,12.175,-64.025,172.881,24.044,154.329
C02524=1071.134,12.425,-64.040,172.882,24.046,154.329
C02525=1071.141,12.674,-64.055,172.884,24.048,154.330
C02526=1071.146,12.924,-64.068,172.885,24.051,154.330
C02527=1071.153,13.174,-64.083,172.886,24.054,154.330
C02528=1071.159,13.423,-64.098,172.887,24.056,154.331
C02529=1071.165,13.672,-64.113,172.889,24.058,154.331
C02530=1071.171,13.922,-64.128,172.890,24.061,154.331
C02531=1071.177,14.203,-64.144,172.891,24.064,154.332
C02532=1071.184,14.484,-64.161,172.894,24.067,154.332
C02533=1071.191,14.765,-64.178,172.895,24.069,154.332
C02534=1071.198,15.045,-64.195,172.896,24.072,154.333
C02535=1071.203,15.295,-64.209,172.898,24.075,154.333
C02536=1071.209,15.545,-64.224,172.900,24.078,154.333
C02537=1071.215,15.795,-64.239,172.901,24.081,154.334
C02538=1071.221,16.044,-64.254,172.902,24.083,154.334
C02539=1071.227,16.293,-64.269,172.903,24.085,154.334
C02540=1071.232,16.542,-64.284,172.905,24.088,154.335
C02541=1071.239,16.792,-64.299,172.906,24.091,154.335
C02542=1071.245,17.042,-64.314,172.907,24.093,154.335
C02543=1071.250,17.291,-64.329,172.909,24.095,154.335
C02544=1071.257,17.541,-64.344,172.910,24.098,154.336
C02545=1071.262,17.790,-64.358,172.911,24.101,154.336
C02546=1071.269,18.039,-64.373,172.913,24.103,154.336
C02547=1071.274,18.289,-64.389,172.915,24.106,154.337
C02548=1071.280,18.538,-64.403,172.916,24.109,154.337
C02549=1071.287,18.788,-64.418,172.917,24.111,154.337
C02550=1071.292,19.037,-64.434,172.919,24.114,154.338
C02551=1071.298,19.287,-64.449,172.920,24.117,154.338
C02552=1071.304,19.536,-64.463,172.921,24.119,154.338
C02553=1071.309,19.786,-64.479,172.923,24.121,154.339
C02554=1071.316,20.035,-64.494,172.924,24.124,154.339
C02555=1071.322,20.285,-64.509,172.925,24.127,154.339
C02556=1071.327,20.534,-64.524,172.927,24.129,154.340
C02557=1071.334,20.784,-64.539,172.928,24.131,154.340
C02558=1071.340,21.034,-64.554,172.929,24.134,154.340
C02559=1071.345,21.283,-64.569,172.931,24.137,154.340
C02560=1071.351,21.533,-64.584,172.933,24.139,154.341
C02561=1071.357,21.782,-64.600,172.934,24.142,154.341
C02562=1071.363,22.031,-64.615,172.935,24.145,154.341
C02563=1071.370,22.280,-64.630,172.937,24.147,154.342
C02564=1071.375,22.530,-64.645,172.938,24.150,154.342
C02565=1071.381,22.779,-64.660,172.939,24.152,154.342
C02566=1071.387,23.029,-64.675,172.941,24.155,154.343
C02567=1071.392,23.278,-64.690,172.942,24.158,154.343
C02568=1071.398,23.528,-64.706,172.943,24.160,154.343
C02569=1071.405,23.777,-64.721,172.944,24.163,154.344
C02570=1071.411,24.027,-64.736,172.946,24.166,154.344
C02571=1071.416,24.276,-64.751,172.947,24.168,154.344
C02572=1071.423,24.526,-64.766,172.949,24.171,154.345
C02573=1071.428,24.776,-64.782,172.950,24.174,154.345
C02574=1071.434,25.024,-64.797,172.952,24.176,154.345
C02575=1071.440,25.274,-64.812,172.953,24.178,154.346
C02576=1071.446,25.524,-64.827,172.954,24.181,154.346
C02577=1071.451,25.773,-64.843,172.956,24.184,154.346
C02578=1071.458,26.022,-64.858,172.957,24.186,154.347
C02579=1071.464,26.272,-64.874,172.958,24.189,154.347
C02580=1071.470,26.522,-64.889,172.960,24.191,154.347
C02581=1071.476,26.771,-64.903,172.961,24.194,154.348
C02582=1071.482,27.020,-64.920,172.962,24.197,154.348
C02583=1071.487,27.270,-64.935,172.964,24.199,154.348
C02584=1071.494,27.520,-64.950,172.966,24.202,154.348
C02585=1071.499,27.769,-64.965,172.967,24.205,154.349
C02586=1071.506,28.018,-64.981,172.968,24.207,154.349
C02587=1071.511,28.268,-64.996,172.970,24.209,154.349
C02588=1071.518,28.518,-65.011,172.971,24.212,154.350
C02589=1071.523,28.766,-65.027,172.972,24.215,154.350
C02590=1071.529,29.016,-65.042,172.974,24.217,154.350
C02591=1071.535,29.266,-65.058,172.975,24.220,154.351
C02592=1071.541,29.515,-65.074,172.976,24.222,154.351
C02593=1071.547,29.764,-65.089,172.977,24.225,154.351
C02594=1071.552,30.014,-65.104,172.979,24.228,154.352
C02595=1071.559,30.296,-65.122,172.981,24.231,154.352
C02596=1071.566,30.579,-65.139,172.982,24.234,154.353
C02597=1071.572,30.861,-65.157,172.984,24.237,154.353
C02598=1071.578,31.143,-65.174,172.986,24.240,154.353
C02599=1071.585,31.392,-65.190,172.987,24.243,154.354
C02600=1071.591,31.642,-65.206,172.988,24.245,154.354
C02601=1071.596,31.892,-65.221,172.989,24.248,154.354
C02602=1071.603,32.140,-65.237,172.991,24.250,154.355
C02603=1071.608,32.390,-65.252,172.992,24.253,154.355
C02604=1071.614,32.640,-65.268,172.993,24.256,154.355
C02605=1071.621,32.889,-65.283,172.996,24.258,154.355
C02606=1071.626,33.139,-65.300,172.997,24.261,154.356
C02607=1071.632,33.388,-65.315,172.998,24.264,154.356
C02608=1071.638,33.637,-65.330,173.000,24.266,154.356
C02609=1071.644,33.887,-65.346,173.001,24.269,154.357
C02610=1071.650,34.136,-65.362,173.002,24.271,154.357
C02611=1071.656,34.386,-65.377,173.003,24.274,154.357
C02612=1071.662,34.635,-65.393,173.005,24.277,154.358
C02613=1071.667,34.885,-65.409,173.006,24.279,154.358
C02614=1071.673,35.134,-65.425,173.007,24.281,154.358
C02615=1071.680,35.384,-65.440,173.010,24.285,154.359
C02616=1071.685,35.633,-65.456,173.011,24.287,154.359
C02617=1071.691,35.883,-65.472,173.012,24.290,154.359
C02618=1071.698,36.132,-65.487,173.013,24.292,154.360
C02619=1071.703,36.381,-65.502,173.015,24.295,154.360
C02620=1071.709,36.631,-65.519,173.016,24.298,154.360
C02621=1071.715,36.880,-65.535,173.017,24.300,154.361
C02622=1071.721,37.130,-65.550,173.019,24.302,154.361
C02623=1071.727,37.379,-65.566,173.020,24.305,154.361
C02624=1071.733,37.629,-65.582,173.021,24.308,154.362
C02625=1071.739,37.878,-65.598,173.023,24.311,154.362
C02626=1071.745,38.127,-65.614,173.025,24.313,154.362
C02627=1071.750,38.377,-65.629,173.026,24.316,154.363
C02628=1071.756,38.626,-65.645,173.027,24.319,154.363
C02629=1071.762,38.876,-65.661,173.029,24.321,154.363
C02630=1071.768,39.125,-65.677,173.030,24.324,154.364
C02631=1071.774,39.375,-65.693,173.031,24.326,154.364
C02632=1071.780,39.625,-65.709,173.033,24.329,154.364
C02633=1071.785,39.873,-65.724,173.034,24.332,154.365
C02634=1071.791,40.123,-65.741,173.035,24.335,154.365
C02635=1071.798,40.372,-65.756,173.037,24.337,154.365
C02636=1071.803,40.622,-65.772,173.039,24.340,154.366
C02637=1071.809,40.871,-65.788,173.040,24.343,154.366
C02638=1071.815,41.120,-65.804,173.041,24.345,154.366
C02639=1071.821,41.370,-65.820,173.043,24.348,154.367
C02640=1071.827,41.620,-65.836,173.044,24.350,154.367
C02641=1071.833,41.869,-65.852,173.045,24.353,154.367
C02642=1071.838,42.118,-65.868,173.047,24.356,154.368
C02643=1071.844,42.368,-65.884,173.048,24.358,154.368
C02644=1071.850,42.617,-65.900,173.049,24.361,154.368
C02645=1071.856,42.866,-65.916,173.051,24.363,154.369
C02646=1071.861,43.116,-65.933,173.053,24.367,154.369
C02647=1071.867,43.366,-65.948,173.054,24.369,154.369
C02648=1071.873,43.615,-65.964,173.055,24.372,154.370
C02649=1071.879,43.864,-65.981,173.057,24.374,154.370
C02650=1071.885,44.114,-65.997,173.058,24.377,154.370
C02651=1071.891,44.363,-66.013,173.059,24.379,154.371
C02652=1071.897,44.613,-66.029,173.060,24.382,154.371
C02653=1071.902,44.862,-66.045,173.062,24.385,154.371
C02654=1071.908,45.111,-66.061,173.063,24.388,154.372
C02655=1071.914,45.360,-66.077,173.065,24.390,154.372
C02656=1071.920,45.610,-66.093,173.067,24.393,154.372
C02657=1071.925,45.859,-66.110,173.068,24.396,154.373
C02658=1071.931,46.109,-66.127,173.069,24.399,154.373
C02659=1071.938,46.391,-66.145,173.070,24.402,154.374
C02660=1071.944,46.673,-66.163,173.072,24.405,154.374
C02661=1071.950,46.956,-66.182,173.074,24.408,154.374
C02662=1071.957,47.238,-66.200,173.075,24.411,154.375
C02663=1071.963,47.487,-66.216,173.076,24.413,154.375
C02664=1071.969,47.736,-66.232,173.078,24.416,154.375
C02665=1071.974,47.986,-66.248,173.080,24.419,154.376
C02666=1071.980,48.236,-66.264,173.081,24.422,154.376
C02667=1071.986,48.485,-66.281,173.082,24.424,154.376
C02668=1071.991,48.735,-66.297,173.084,24.427,154.377
C02669=1071.997,48.984,-66.314,173.085,24.429,154.377
C02670=1072.003,49.233,-66.330,173.086,24.432,154.377
C02671=1072.009,49.483,-66.346,173.088,24.435,154.378
C02672=1072.015,49.732,-66.363,173.089,24.437,154.378
C02673=1072.021,49.982,-66.379,173.091,24.440,154.378
C02674=1072.026,50.231,-66.395,173.092,24.443,154.379
C02675=1072.032,50.480,-66.412,173.094,24.445,154.379
C02676=1072.038,50.730,-66.428,173.095,24.448,154.379
C02677=1072.044,50.979,-66.444,173.096,24.451,154.380
C02678=1072.050,51.229,-66.461,173.098,24.454,154.380
C02679=1072.055,51.478,-66.477,173.099,24.456,154.380
C02680=1072.061,51.728,-66.494,173.100,24.459,154.381
C02681=1072.068,51.976,-66.511,173.101,24.461,154.381
C02682=1072.073,52.226,-66.527,173.104,24.464,154.381
C02683=1072.079,52.475,-66.544,173.105,24.467,154.382
C02684=1072.085,52.725,-66.560,173.106,24.469,154.382
C02685=1072.091,52.974,-66.576,173.108,24.472,154.382
C02686=1072.097,53.223,-66.592,173.109,24.475,154.383
C02687=1072.102,53.473,-66.609,173.110,24.477,154.383
C02688=1072.108,53.722,-66.626,173.112,24.480,154.383
C02689=1072.114,53.972,-66.642,173.113,24.483,154.384
C02690=1072.120,54.221,-66.658,173.115,24.485,154.384
C02691=1072.125,54.470,-66.676,173.116,24.488,154.384
C02692=1072.131,54.719,-66.692,173.118,24.491,154.385
C02693=1072.138,54.969,-66.709,173.119,24.493,154.385
C02694=1072.144,55.219,-66.725,173.120,24.496,154.385
C02695=1072.149,55.468,-66.742,173.122,24.498,154.386
C02696=1072.155,55.718,-66.758,173.123,24.501,154.386
C02697=1072.161,55.967,-66.775,173.124,24.504,154.386
C02698=1072.167,56.216,-66.791,173.126,24.507,154.387
C02699=1072.172,56.466,-66.808,173.128,24.509,154.387
C02700=1072.178,56.715,-66.824,173.129,24.512,154.387
C02701=1072.184,56.964,-66.840,173.130,24.515,154.388
C02702=1072.190,57.213,-66.857,173.132,24.517,154.388
C02703=1072.196,57.463,-66.875,173.133,24.520,154.388
C02704=1072.202,57.713,-66.891,173.134,24.522,154.389
C02705=1072.208,57.962,-66.907,173.136,24.525,154.389
C02706=1072.214,58.211,-66.925,173.138,24.528,154.389
C02707=1072.220,58.460,-66.941,173.139,24.530,154.390
C02708=1072.226,58.710,-66.957,173.141,24.533,154.390
C02709=1072.232,58.958,-66.974,173.142,24.535,154.390
C02710=1072.238,59.209,-66.991,173.143,24.538,154.391
C02711=1072.244,59.458,-67.008,173.145,24.541,154.391
C02712=1072.250,59.708,-67.024,173.146,24.543,154.391
C02713=1072.255,59.957,-67.042,173.147,24.546,154.392
C02714=1072.261,60.206,-67.058,173.150,24.549,154.392
C02715=1072.268,60.456,-67.074,173.151,24.552,154.392
C02716=1072.274,60.705,-67.091,173.152,24.554,154.393
C02717=1072.279,60.954,-67.108,173.154,24.556,154.393
C02718=1072.285,61.204,-67.124,173.155,24.559,154.393
C02719=1072.291,61.452,-67.141,173.156,24.562,154.394
C02720=1072.297,61.703,-67.159,173.157,24.564,154.394
C02721=1072.303,61.952,-67.176,173.159,24.567,154.394
C02722=1072.309,62.201,-67.192,173.161,24.570,154.395
C02723=1072.316,62.483,-67.212,173.162,24.572,154.395
C02724=1072.323,62.766,-67.230,173.164,24.575,154.395
C02725=1072.329,63.047,-67.249,173.166,24.579,154.396
C02726=1072.336,63.329,-67.268,173.167,24.582,154.396
C02727=1072.342,63.578,-67.285,173.168,24.584,154.396
C02728=1072.348,63.828,-67.303,173.171,24.587,154.397
C02729=1072.354,64.078,-67.319,173.172,24.589,154.397
C02730=1072.360,64.326,-67.336,173.173,24.592,154.397
C02731=1072.365,64.576,-67.353,173.175,24.594,154.398
C02732=1072.372,64.825,-67.370,173.176,24.597,154.398
C02733=1072.378,65.075,-67.387,173.177,24.599,154.398
C02734=1072.384,65.324,-67.404,173.178,24.602,154.399
C02735=1072.389,65.573,-67.421,173.181,24.605,154.399
C02736=1072.395,65.822,-67.438,173.182,24.608,154.399
C02737=1072.401,66.072,-67.455,173.183,24.610,154.400
C02738=1072.407,66.322,-67.472,173.185,24.613,154.400
C02739=1072.413,66.571,-67.489,173.186,24.616,154.400
C02740=1072.418,66.820,-67.506,173.187,24.618,154.401
C02741=1072.425,67.070,-67.523,173.189,24.621,154.401
C02742=1072.430,67.319,-67.540,173.191,24.624,154.401
C02743=1072.435,67.569,-67.557,173.192,24.626,154.402
C02744=1072.442,67.817,-67.574,173.194,24.629,154.402
C02745=1072.448,68.067,-67.592,173.195,24.632,154.402
C02746=1072.454,68.316,-67.608,173.196,24.634,154.403
C02747=1072.459,68.565,-67.626,173.197,24.637,154.403
C02748=1072.464,68.815,-67.643,173.199,24.639,154.403
C02749=1072.471,69.065,-67.660,173.201,24.643,154.404
C02750=1072.477,69.314,-67.678,173.202,24.645,154.404
C02751=1072.483,69.563,-67.694,173.204,24.647,154.404
C02752=1072.488,69.812,-67.712,173.205,24.650,154.405
C02753=1072.494,70.062,-67.730,173.206,24.653,154.405
C02754=1072.500,70.311,-67.746,173.208,24.655,154.406
C02755=1072.506,70.560,-67.763,173.209,24.658,154.406
C02756=1072.511,70.809,-67.781,173.211,24.661,154.406
C02757=1072.517,71.060,-67.798,173.213,24.663,154.406
C02758=1072.523,71.308,-67.815,173.214,24.666,154.407
C02759=1072.529,71.557,-67.833,173.215,24.669,154.407
C02760=1072.535,71.808,-67.850,173.217,24.672,154.408
C02761=1072.540,72.057,-67.867,173.218,24.674,154.408
C02762=1072.547,72.305,-67.884,173.219,24.677,154.408
C02763=1072.552,72.554,-67.902,173.221,24.679,154.408
C02764=1072.558,72.805,-67.919,173.223,24.682,154.409
C02765=1072.563,73.054,-67.937,173.224,24.685,154.409
C02766=1072.570,73.303,-67.954,173.225,24.688,154.410
C02767=1072.576,73.552,-67.972,173.227,24.690,154.410
C02768=1072.581,73.802,-67.989,173.228,24.692,154.410
C02769=1072.587,74.051,-68.006,173.230,24.696,154.411
C02770=1072.593,74.300,-68.023,173.232,24.698,154.411
C02771=1072.599,74.550,-68.041,173.233,24.701,154.411
C02772=1072.604,74.799,-68.059,173.234,24.703,154.412
C02773=1072.610,75.049,-68.076,173.236,24.706,154.412
C02774=1072.616,75.298,-68.093,173.237,24.708,154.412
C02775=1072.622,75.547,-68.110,173.239,24.712,154.413
C02776=1072.628,75.796,-68.128,173.241,24.714,154.413
C02777=1072.634,76.045,-68.146,173.242,24.716,154.413
C02778=1072.639,76.295,-68.163,173.243,24.719,154.414
C02779=1072.645,76.545,-68.181,173.245,24.722,154.414
C02780=1072.651,76.794,-68.198,173.246,24.724,154.414
C02781=1072.657,77.043,-68.215,173.248,24.727,154.414
C02782=1072.663,77.292,-68.233,173.249,24.730,154.415
C02783=1072.668,77.541,-68.251,173.251,24.732,154.415
C02784=1072.674,77.791,-68.269,173.252,24.735,154.415
C02785=1072.680,78.040,-68.286,173.253,24.738,154.416
C02786=1072.686,78.289,-68.304,173.255,24.740,154.416
C02787=1072.692,78.571,-68.323,173.257,24.743,154.417
C02788=1072.699,78.854,-68.343,173.258,24.746,154.417
C02789=1072.705,79.135,-68.363,173.260,24.749,154.417
C02790=1072.712,79.418,-68.383,173.262,24.752,154.418
C02791=1072.717,79.667,-68.401,173.263,24.755,154.418
C02792=1072.724,79.916,-68.419,173.265,24.758,154.418
C02793=1072.729,80.165,-68.436,173.267,24.761,154.419
C02794=1072.735,80.414,-68.454,173.268,24.763,154.419
C02795=1072.741,80.664,-68.472,173.269,24.766,154.419
C02796=1072.746,80.913,-68.489,173.271,24.768,154.420
C02797=1072.752,81.162,-68.507,173.272,24.771,154.420
C02798=1072.758,81.412,-68.525,173.274,24.774,154.420
C02799=1072.763,81.661,-68.542,173.276,24.776,154.421
C02800=1072.770,81.911,-68.560,173.277,24.779,154.421
C02801=1072.775,82.160,-68.578,173.278,24.782,154.421
C02802=1072.781,82.409,-68.595,173.279,24.784,154.422
C02803=1072.787,82.659,-68.613,173.281,24.787,154.422
C02804=1072.793,82.907,-68.632,173.283,24.790,154.422
C02805=1072.799,83.157,-68.650,173.284,24.792,154.423
C02806=1072.804,83.406,-68.667,173.286,24.795,154.423
C02807=1072.810,83.655,-68.685,173.287,24.798,154.423
C02808=1072.816,83.905,-68.703,173.288,24.800,154.424
C02809=1072.821,84.154,-68.720,173.291,24.803,154.424
C02810=1072.827,84.403,-68.738,173.292,24.806,154.425
C02811=1072.832,84.653,-68.756,173.293,24.808,154.425
C02812=1072.838,84.902,-68.774,173.295,24.811,154.425
C02813=1072.844,85.151,-68.793,173.296,24.814,154.426
C02814=1072.850,85.401,-68.810,173.297,24.816,154.426
C02815=1072.856,85.650,-68.828,173.300,24.819,154.426
C02816=1072.862,85.899,-68.846,173.301,24.822,154.426
C02817=1072.867,86.148,-68.864,173.302,24.824,154.427
C02818=1072.874,86.398,-68.882,173.304,24.827,154.427
C02819=1072.879,86.647,-68.900,173.305,24.829,154.427
C02820=1072.885,86.896,-68.918,173.307,24.832,154.428
C02821=1072.891,87.145,-68.935,173.309,24.835,154.428
C02822=1072.897,87.395,-68.953,173.310,24.838,154.429
C02823=1072.902,87.644,-68.972,173.311,24.840,154.429
C02824=1072.908,87.894,-68.990,173.313,24.842,154.429
C02825=1072.914,88.143,-69.008,173.315,24.845,154.429
C02826=1072.920,88.392,-69.026,173.316,24.848,154.430
C02827=1072.926,88.604,-69.041,173.318,24.850,154.430
C02828=1072.930,88.816,-69.056,173.319,24.852,154.430
C02829=1072.935,89.029,-69.071,173.320,24.854,154.431
C02830=1072.940,89.241,-69.088,173.321,24.857,154.431
C02831=1072.946,89.454,-69.103,173.322,24.859,154.431
C02832=1072.950,89.666,-69.118,173.324,24.861,154.431
C02833=1072.955,89.878,-69.133,173.325,24.863,154.432
C02834=1072.960,90.091,-69.149,173.327,24.866,154.432
C02835=1072.966,90.340,-69.166,173.328,24.868,154.432
C02836=1072.972,90.589,-69.184,173.329,24.871,154.433
C02837=1072.978,90.838,-69.203,173.331,24.873,154.433
C02838=1072.983,91.088,-69.221,173.333,24.876,154.433
C02839=1072.989,91.337,-69.240,173.334,24.879,154.434
C02840=1072.995,91.586,-69.257,173.336,24.882,154.434
C02841=1073.000,91.836,-69.276,173.337,24.884,154.434
C02842=1073.006,92.084,-69.294,173.338,24.887,154.435
C02843=1073.012,92.334,-69.312,173.341,24.890,154.435
C02844=1073.017,92.584,-69.330,173.342,24.892,154.435
C02845=1073.023,92.833,-69.349,173.343,24.895,154.436
C02846=1073.029,93.082,-69.367,173.345,24.897,154.436
C02847=1073.035,93.331,-69.386,173.346,24.900,154.436
C02848=1073.040,93.580,-69.403,173.348,24.903,154.437
C02849=1073.047,93.829,-69.422,173.350,24.905,154.437
C02850=1073.052,94.079,-69.441,173.351,24.908,154.437
C02851=1073.060,94.435,-69.467,173.353,24.912,154.438
C02852=1073.068,94.791,-69.493,173.355,24.915,154.438
C02853=1073.077,95.146,-69.519,173.358,24.920,154.439
C02854=1073.085,95.502,-69.545,173.360,24.923,154.439
C02855=1073.090,95.751,-69.564,173.362,24.926,154.440
C02856=1073.096,96.001,-69.582,173.363,24.928,154.440
C02857=1073.103,96.250,-69.600,173.364,24.931,154.440
C02858=1073.107,96.499,-69.619,173.367,24.933,154.440
C02859=1073.114,96.748,-69.637,173.368,24.936,154.441
C02860=1073.119,96.998,-69.655,173.369,24.939,154.441
C02861=1073.125,97.247,-69.674,173.371,24.942,154.442
C02862=1073.131,97.497,-69.692,173.373,24.944,154.442
C02863=1073.136,97.745,-69.711,173.374,24.947,154.442
C02864=1073.143,97.995,-69.730,173.376,24.949,154.443
C02865=1073.148,98.245,-69.748,173.377,24.952,154.443
C02866=1073.154,98.493,-69.766,173.378,24.954,154.443
C02867=1073.160,98.743,-69.784,173.381,24.957,154.443
C02868=1073.166,98.992,-69.804,173.382,24.960,154.444
C02869=1073.172,99.241,-69.822,173.383,24.963,154.444
C02870=1073.177,99.491,-69.840,173.385,24.965,154.444
C02871=1073.183,99.740,-69.859,173.387,24.968,154.445
C02872=1073.188,99.989,-69.878,173.388,24.970,154.445
C02873=1073.195,100.238,-69.896,173.390,24.973,154.445
C02874=1073.201,100.487,-69.914,173.391,24.975,154.446
C02875=1073.206,100.736,-69.933,173.393,24.978,154.446
C02876=1073.212,100.986,-69.951,173.395,24.981,154.446
C02877=1073.218,101.235,-69.971,173.396,24.983,154.447
C02878=1073.224,101.484,-69.989,173.397,24.986,154.447
C02879=1073.229,101.734,-70.007,173.400,24.989,154.447
C02880=1073.235,101.983,-70.027,173.401,24.991,154.448
C02881=1073.241,102.232,-70.045,173.402,24.994,154.448
C02882=1073.246,102.481,-70.064,173.404,24.997,154.448
C02883=1073.252,102.731,-70.083,173.405,24.999,154.449
C02884=1073.257,102.980,-70.101,173.407,25.002,154.449
C02885=1073.263,103.229,-70.120,173.409,25.004,154.449
C02886=1073.270,103.478,-70.139,173.410,25.007,154.450
C02887=1073.275,103.727,-70.158,173.411,25.010,154.450
C02888=1073.280,103.977,-70.176,173.414,25.012,154.450
C02889=1073.286,104.226,-70.195,173.415,25.015,154.451
C02890=1073.292,104.475,-70.214,173.416,25.018,154.451
C02891=1073.297,104.724,-70.233,173.418,25.020,154.451
C02892=1073.304,104.973,-70.252,173.420,25.023,154.452
C02893=1073.309,105.223,-70.271,173.421,25.025,154.452
C02894=1073.314,105.472,-70.289,173.423,25.028,154.452
C02895=1073.321,105.721,-70.308,173.424,25.031,154.453
C02896=1073.326,105.971,-70.327,173.426,25.033,154.453
C02897=1073.332,106.220,-70.346,173.428,25.036,154.453
C02898=1073.338,106.468,-70.364,173.429,25.038,154.454
C02899=1073.343,106.718,-70.384,173.432,25.041,154.454
C02900=1073.349,106.967,-70.403,173.433,25.044,154.454
C02901=1073.356,107.216,-70.422,173.434,25.046,154.455
C02902=1073.361,107.465,-70.440,173.436,25.049,154.455
C02903=1073.366,107.715,-70.460,173.438,25.052,154.455
C02904=1073.372,107.965,-70.478,173.439,25.054,154.455
C02905=1073.378,108.214,-70.497,173.441,25.057,154.456
C02906=1073.384,108.463,-70.516,173.442,25.059,154.456
C02907=1073.389,108.712,-70.535,173.444,25.062,154.456
C02908=1073.395,108.961,-70.554,173.446,25.064,154.457
C02909=1073.401,109.211,-70.573,173.447,25.067,154.457
C02910=1073.407,109.460,-70.592,173.448,25.070,154.457
C02911=1073.413,109.709,-70.611,173.451,25.072,154.458
C02912=1073.418,109.958,-70.630,173.452,25.075,154.458
C02913=1073.424,110.207,-70.649,173.453,25.077,154.458
C02914=1073.430,110.457,-70.668,173.456,25.080,154.459
C02915=1073.437,110.739,-70.690,173.457,25.083,154.459
C02916=1073.443,111.021,-70.711,173.459,25.086,154.459
C02917=1073.450,111.303,-70.733,173.461,25.089,154.460
C02918=1073.456,111.584,-70.754,173.463,25.092,154.460
C02919=1073.461,111.834,-70.774,173.464,25.095,154.460
C02920=1073.468,112.083,-70.792,173.466,25.097,154.461
C02921=1073.474,112.332,-70.812,173.468,25.100,154.461
C02922=1073.480,112.581,-70.831,173.469,25.102,154.461
C02923=1073.485,112.830,-70.850,173.471,25.105,154.462
C02924=1073.490,113.079,-70.870,173.473,25.108,154.462
C02925=1073.496,113.329,-70.889,173.474,25.110,154.462
C02926=1073.502,113.578,-70.908,173.476,25.113,154.463
C02927=1073.508,113.827,-70.927,173.477,25.115,154.463
C02928=1073.514,114.076,-70.947,173.479,25.118,154.463
C02929=1073.520,114.326,-70.966,173.481,25.120,154.464
C02930=1073.525,114.574,-70.985,173.482,25.123,154.464
C02931=1073.531,114.824,-71.004,173.484,25.126,154.464
C02932=1073.536,115.073,-71.023,173.486,25.129,154.465
C02933=1073.542,115.323,-71.042,173.487,25.131,154.465
C02934=1073.548,115.572,-71.062,173.489,25.133,154.465
C02935=1073.552,115.821,-71.082,173.491,25.137,154.466
C02936=1073.558,116.070,-71.101,173.492,25.139,154.466
C02937=1073.564,116.319,-71.120,173.494,25.142,154.466
C02938=1073.570,116.568,-71.140,173.496,25.145,154.467
C02939=1073.575,116.818,-71.160,173.497,25.147,154.467
C02940=1073.581,117.067,-71.179,173.499,25.150,154.467
C02941=1073.586,117.316,-71.198,173.501,25.152,154.468
C02942=1073.592,117.565,-71.218,173.502,25.155,154.468
C02943=1073.598,117.814,-71.237,173.504,25.158,154.468
C02944=1073.604,118.064,-71.256,173.505,25.160,154.469
C02945=1073.610,118.312,-71.276,173.507,25.163,154.469
C02946=1073.615,118.562,-71.295,173.509,25.165,154.469
C02947=1073.620,118.812,-71.315,173.510,25.168,154.470
C02948=1073.626,119.060,-71.335,173.512,25.171,154.470
C02949=1073.631,119.309,-71.354,173.514,25.173,154.470
C02950=1073.637,119.558,-71.373,173.515,25.176,154.471
C02951=1073.643,119.807,-71.393,173.517,25.179,154.471
C02952=1073.649,120.057,-71.412,173.519,25.182,154.471
C02953=1073.654,120.306,-71.432,173.520,25.184,154.472
C02954=1073.660,120.555,-71.452,173.522,25.187,154.472
C02955=1073.666,120.804,-71.471,173.524,25.189,154.472
C02956=1073.671,121.054,-71.491,173.525,25.192,154.472
C02957=1073.677,121.303,-71.511,173.528,25.194,154.473
C02958=1073.683,121.552,-71.531,173.529,25.197,154.473
C02959=1073.689,121.801,-71.550,173.530,25.200,154.473
C02960=1073.694,122.051,-71.569,173.532,25.202,154.474
C02961=1073.700,122.299,-71.589,173.534,25.205,154.474
C02962=1073.705,122.548,-71.608,173.535,25.207,154.474
C02963=1073.711,122.797,-71.629,173.537,25.210,154.475
C02964=1073.716,123.047,-71.648,173.539,25.213,154.475
C02965=1073.722,123.296,-71.668,173.540,25.215,154.475
C02966=1073.728,123.545,-71.687,173.542,25.217,154.476
C02967=1073.734,123.794,-71.707,173.544,25.221,154.476
C02968=1073.740,124.043,-71.726,173.546,25.223,154.476
C02969=1073.745,124.292,-71.747,173.547,25.225,154.477
C02970=1073.751,124.542,-71.766,173.549,25.228,154.477
C02971=1073.757,124.791,-71.786,173.551,25.231,154.477
C02972=1073.763,125.039,-71.806,173.552,25.233,154.478
C02973=1073.768,125.289,-71.825,173.554,25.236,154.478
C02974=1073.774,125.538,-71.845,173.556,25.239,154.478
C02975=1073.779,125.787,-71.865,173.557,25.241,154.479
C02976=1073.785,126.036,-71.885,173.559,25.244,154.479
C02977=1073.791,126.286,-71.904,173.561,25.246,154.479
C02978=1073.798,126.535,-71.924,173.563,25.249,154.479
C02979=1073.803,126.817,-71.947,173.565,25.251,154.480
C02980=1073.810,127.099,-71.969,173.567,25.255,154.480
C02981=1073.816,127.381,-71.992,173.569,25.258,154.480
C02982=1073.824,127.662,-72.014,173.570,25.260,154.481
C02983=1073.829,127.912,-72.034,173.573,25.263,154.481
C02984=1073.835,128.161,-72.054,173.574,25.266,154.481
C02985=1073.841,128.410,-72.074,173.576,25.268,154.482
C02986=1073.846,128.659,-72.093,173.578,25.271,154.482
C02987=1073.852,128.908,-72.114,173.579,25.273,154.482
C02988=1073.858,129.157,-72.134,173.581,25.276,154.483
C02989=1073.864,129.407,-72.153,173.583,25.278,154.483
C02990=1073.870,129.656,-72.173,173.584,25.281,154.483
C02991=1073.876,129.905,-72.193,173.586,25.283,154.484
C02992=1073.881,130.154,-72.214,173.588,25.286,154.484
C02993=1073.887,130.404,-72.233,173.590,25.288,154.484
C02994=1073.893,130.652,-72.253,173.592,25.291,154.484
C02995=1073.899,130.901,-72.273,173.593,25.293,154.485
C02996=1073.904,131.150,-72.294,173.595,25.296,154.485
C02997=1073.910,131.400,-72.313,173.597,25.299,154.485
C02998=1073.916,131.649,-72.333,173.598,25.301,154.486
C02999=1073.922,131.898,-72.353,173.600,25.304,154.486
C03000=1073.928,132.147,-72.374,173.602,25.306,154.486
C03001=1073.934,132.396,-72.394,173.604,25.309,154.487
C03002=1073.939,132.646,-72.414,173.606,25.312,154.487
C03003=1073.945,132.895,-72.433,173.607,25.314,154.487
C03004=1073.950,133.144,-72.454,173.609,25.316,154.487
C03005=1073.956,133.392,-72.474,173.611,25.319,154.488
C03006=1073.962,133.642,-72.495,173.612,25.322,154.488
C03007=1073.968,133.891,-72.515,173.614,25.324,154.488
C03008=1073.973,134.140,-72.535,173.616,25.327,154.489
C03009=1073.979,134.389,-72.555,173.618,25.330,154.489
C03010=1073.984,134.639,-72.575,173.620,25.332,154.489
C03011=1073.990,134.888,-72.595,173.621,25.334,154.490
C03012=1073.995,135.137,-72.616,173.623,25.337,154.490
C03013=1074.001,135.386,-72.636,173.625,25.340,154.490
C03014=1074.007,135.635,-72.657,173.626,25.342,154.491
C03015=1074.013,135.884,-72.677,173.629,25.345,154.491
C03016=1074.018,136.133,-72.697,173.630,25.348,154.491
C03017=1074.024,136.382,-72.717,173.632,25.350,154.492
C03018=1074.029,136.631,-72.738,173.634,25.353,154.492
C03019=1074.035,136.880,-72.758,173.635,25.356,154.492
C03020=1074.041,137.130,-72.779,173.638,25.358,154.492
C03021=1074.047,137.379,-72.798,173.639,25.360,154.493
C03022=1074.053,137.628,-72.819,173.641,25.363,154.493
C03023=1074.059,137.877,-72.839,173.643,25.366,154.493
C03024=1074.064,138.126,-72.860,173.644,25.368,154.494
C03025=1074.070,138.376,-72.880,173.647,25.371,154.494
C03026=1074.076,138.624,-72.900,173.648,25.373,154.494
C03027=1074.081,138.874,-72.921,173.649,25.376,154.495
C03028=1074.087,139.122,-72.941,173.652,25.379,154.495
C03029=1074.092,139.371,-72.962,173.653,25.381,154.495
C03030=1074.098,139.621,-72.983,173.655,25.384,154.495
C03031=1074.104,139.869,-73.003,173.657,25.386,154.496
C03032=1074.110,140.119,-73.024,173.659,25.389,154.496
C03033=1074.116,140.367,-73.044,173.661,25.391,154.496
C03034=1074.121,140.617,-73.065,173.662,25.394,154.497
C03035=1074.127,140.866,-73.085,173.664,25.397,154.497
C03036=1074.132,141.115,-73.106,173.666,25.399,154.497
C03037=1074.138,141.364,-73.126,173.668,25.402,154.498
C03038=1074.143,141.613,-73.147,173.670,25.404,154.498
C03039=1074.149,141.863,-73.168,173.671,25.407,154.498
C03040=1074.155,142.112,-73.188,173.673,25.410,154.499
C03041=1074.161,142.361,-73.208,173.675,25.412,154.499
C03042=1074.166,142.609,-73.230,173.677,25.415,154.499
C03043=1074.172,142.891,-73.252,173.679,25.418,154.500
C03044=1074.179,143.173,-73.276,173.681,25.421,154.500
C03045=1074.185,143.455,-73.300,173.683,25.424,154.500
C03046=1074.191,143.737,-73.323,173.685,25.426,154.501
C03047=1074.197,143.987,-73.344,173.687,25.429,154.501
C03048=1074.203,144.235,-73.364,173.689,25.432,154.501
C03049=1074.209,144.484,-73.385,173.690,25.434,154.502
C03050=1074.215,144.734,-73.406,173.693,25.437,154.502
C03051=1074.220,144.983,-73.427,173.694,25.440,154.502
C03052=1074.226,145.231,-73.447,173.695,25.442,154.503
C03053=1074.231,145.480,-73.468,173.698,25.444,154.503
C03054=1074.237,145.730,-73.489,173.699,25.447,154.503
C03055=1074.243,145.978,-73.510,173.702,25.449,154.503
C03056=1074.248,146.228,-73.531,173.703,25.452,154.504
C03057=1074.255,146.477,-73.551,173.705,25.455,154.504
C03058=1074.260,146.726,-73.572,173.707,25.457,154.504
C03059=1074.266,146.975,-73.593,173.709,25.460,154.505
C03060=1074.271,147.225,-73.614,173.711,25.462,154.505
C03061=1074.277,147.473,-73.635,173.713,25.465,154.505
C03062=1074.283,147.722,-73.655,173.714,25.468,154.505
C03063=1074.289,147.971,-73.677,173.717,25.470,154.506
C03064=1074.294,148.220,-73.697,173.718,25.472,154.506
C03065=1074.300,148.469,-73.718,173.719,25.475,154.506
C03066=1074.306,148.719,-73.739,173.722,25.478,154.507
C03067=1074.311,148.968,-73.760,173.723,25.480,154.507
C03068=1074.317,149.216,-73.781,173.726,25.483,154.507
C03069=1074.322,149.466,-73.802,173.727,25.486,154.508
C03070=1074.328,149.715,-73.823,173.729,25.488,154.508
C03071=1074.334,149.964,-73.844,173.731,25.491,154.508
C03072=1074.339,150.213,-73.865,173.733,25.493,154.508
C03073=1074.345,150.462,-73.886,173.735,25.496,154.509
C03074=1074.351,150.711,-73.908,173.737,25.499,154.509
C03075=1074.356,150.960,-73.928,173.738,25.501,154.509
C03076=1074.362,151.209,-73.949,173.741,25.504,154.510
C03077=1074.368,151.459,-73.970,173.742,25.506,154.510
C03078=1074.373,151.707,-73.992,173.744,25.509,154.510
C03079=1074.379,151.956,-74.013,173.746,25.511,154.511
C03080=1074.385,152.205,-74.034,173.748,25.514,154.511
C03081=1074.390,152.454,-74.055,173.750,25.517,154.511
C03082=1074.396,152.704,-74.076,173.752,25.519,154.512
C03083=1074.401,152.952,-74.097,173.753,25.522,154.512
C03084=1074.407,153.201,-74.119,173.756,25.524,154.512
C03085=1074.413,153.451,-74.140,173.757,25.527,154.512
C03086=1074.418,153.699,-74.161,173.760,25.530,154.513
C03087=1074.425,153.948,-74.182,173.761,25.532,154.513
C03088=1074.430,154.197,-74.203,173.763,25.535,154.513
C03089=1074.436,154.447,-74.225,173.765,25.537,154.514
C03090=1074.442,154.695,-74.246,173.767,25.540,154.514
C03091=1074.447,154.944,-74.266,173.769,25.542,154.514
C03092=1074.453,155.193,-74.288,173.771,25.545,154.515
C03093=1074.459,155.442,-74.309,173.772,25.547,154.515
C03094=1074.464,155.692,-74.330,173.775,25.550,154.515
C03095=1074.469,155.941,-74.352,173.776,25.553,154.516
C03096=1074.475,156.190,-74.374,173.778,25.555,154.516
C03097=1074.481,156.438,-74.395,173.780,25.558,154.516
C03098=1074.487,156.688,-74.416,173.782,25.560,154.516
C03099=1074.492,156.937,-74.437,173.784,25.563,154.517
C03100=1074.498,157.185,-74.458,173.786,25.566,154.517
C03101=1074.503,157.435,-74.481,173.787,25.568,154.517
C03102=1074.509,157.684,-74.501,173.790,25.571,154.518
C03103=1074.515,157.933,-74.523,173.791,25.573,154.518
C03104=1074.520,158.182,-74.544,173.794,25.576,154.518
C03105=1074.527,158.431,-74.566,173.795,25.578,154.519
C03106=1074.531,158.680,-74.588,173.797,25.581,154.519
C03107=1074.539,158.962,-74.611,173.800,25.584,154.519
C03108=1074.545,159.243,-74.636,173.802,25.587,154.520
C03109=1074.552,159.524,-74.660,173.804,25.590,154.520
C03110=1074.557,159.806,-74.684,173.806,25.593,154.520
C03111=1074.564,160.056,-74.706,173.808,25.595,154.520
C03112=1074.568,160.304,-74.728,173.810,25.598,154.521
C03113=1074.575,160.554,-74.749,173.812,25.600,154.521
C03114=1074.580,160.802,-74.771,173.814,25.603,154.521
C03115=1074.586,161.051,-74.792,173.816,25.606,154.522
C03116=1074.592,161.300,-74.814,173.818,25.608,154.522
C03117=1074.597,161.549,-74.836,173.819,25.611,154.522
C03118=1074.603,161.798,-74.857,173.822,25.614,154.523
C03119=1074.608,162.047,-74.879,173.823,25.616,154.523
C03120=1074.614,162.296,-74.901,173.826,25.619,154.523
C03121=1074.619,162.545,-74.923,173.828,25.622,154.524
C03122=1074.625,162.794,-74.944,173.829,25.624,154.524
C03123=1074.630,163.043,-74.966,173.831,25.627,154.524
C03124=1074.636,163.292,-74.988,173.833,25.630,154.525
C03125=1074.641,163.541,-75.010,173.835,25.632,154.525
C03126=1074.646,163.790,-75.032,173.837,25.635,154.525
C03127=1074.652,164.039,-75.053,173.839,25.638,154.525
C03128=1074.657,164.288,-75.075,173.841,25.640,154.526
C03129=1074.663,164.537,-75.097,173.843,25.643,154.526
C03130=1074.668,164.786,-75.119,173.845,25.646,154.526
C03131=1074.674,165.035,-75.140,173.847,25.648,154.527
C03132=1074.679,165.284,-75.162,173.849,25.651,154.527
C03133=1074.685,165.533,-75.184,173.850,25.653,154.527
C03134=1074.690,165.782,-75.206,173.853,25.656,154.528
C03135=1074.696,166.031,-75.228,173.855,25.659,154.528
C03136=1074.701,166.280,-75.250,173.856,25.661,154.528
C03137=1074.707,166.529,-75.272,173.859,25.664,154.529
C03138=1074.713,166.778,-75.294,173.860,25.667,154.529
C03139=1074.718,167.027,-75.316,173.863,25.669,154.529
C03140=1074.724,167.276,-75.338,173.864,25.672,154.530
C03141=1074.729,167.525,-75.360,173.866,25.675,154.530
C03142=1074.734,167.774,-75.382,173.869,25.677,154.530
C03143=1074.740,168.023,-75.403,173.870,25.680,154.530
C03144=1074.746,168.272,-75.426,173.873,25.682,154.531
C03145=1074.752,168.521,-75.448,173.874,25.685,154.531
C03146=1074.757,168.770,-75.470,173.876,25.688,154.531
C03147=1074.762,169.019,-75.492,173.879,25.690,154.532
C03148=1074.769,169.268,-75.514,173.880,25.693,154.532
C03149=1074.773,169.517,-75.536,173.882,25.696,154.532
C03150=1074.780,169.766,-75.558,173.884,25.698,154.533
C03151=1074.784,170.015,-75.580,173.886,25.701,154.533
C03152=1074.790,170.263,-75.603,173.889,25.704,154.533
C03153=1074.796,170.513,-75.624,173.890,25.706,154.534
C03154=1074.801,170.761,-75.646,173.892,25.709,154.534
C03155=1074.808,171.010,-75.668,173.895,25.712,154.534
C03156=1074.813,171.260,-75.691,173.896,25.714,154.535
C03157=1074.818,171.508,-75.713,173.899,25.717,154.535
C03158=1074.824,171.757,-75.735,173.900,25.719,154.535
C03159=1074.830,172.006,-75.757,173.902,25.722,154.535
C03160=1074.835,172.255,-75.780,173.905,25.725,154.536
C03161=1074.841,172.504,-75.801,173.906,25.727,154.536
C03162=1074.846,172.753,-75.824,173.909,25.730,154.536
C03163=1074.852,173.002,-75.847,173.911,25.733,154.537
C03164=1074.858,173.251,-75.868,173.912,25.735,154.537
C03165=1074.863,173.500,-75.891,173.915,25.738,154.537
C03166=1074.869,173.749,-75.913,173.917,25.740,154.537
C03167=1074.875,173.997,-75.935,173.918,25.743,154.538
C03168=1074.880,174.247,-75.957,173.921,25.746,154.538
C03169=1074.886,174.495,-75.980,173.922,25.748,154.538
C03170=1074.892,174.745,-76.002,173.925,25.750,154.539
C03171=1074.898,175.025,-76.027,173.927,25.754,154.539
C03172=1074.905,175.307,-76.052,173.929,25.757,154.539
C03173=1074.910,175.588,-76.078,173.932,25.759,154.540
C03174=1074.917,175.870,-76.103,173.934,25.762,154.540
C03175=1074.924,176.119,-76.125,173.936,25.765,154.540
C03176=1074.928,176.367,-76.147,173.938,25.767,154.541
C03177=1074.934,176.616,-76.170,173.940,25.770,154.541
C03178=1074.940,176.865,-76.192,173.942,25.773,154.541
C03179=1074.946,177.114,-76.215,173.944,25.775,154.542
C03180=1074.952,177.363,-76.238,173.946,25.778,154.542
C03181=1074.957,177.612,-76.260,173.949,25.781,154.542
C03182=1074.963,177.861,-76.282,173.950,25.783,154.542
C03183=1074.969,178.110,-76.305,173.952,25.786,154.543
C03184=1074.974,178.359,-76.327,173.955,25.789,154.543
C03185=1074.980,178.608,-76.350,173.956,25.791,154.543
C03186=1074.986,178.857,-76.372,173.959,25.793,154.544
C03187=1074.991,179.105,-76.394,173.961,25.796,154.544
C03188=1074.997,179.354,-76.417,173.963,25.799,154.544
C03189=1075.003,179.603,-76.440,173.965,25.801,154.545
C03190=1075.009,179.852,-76.462,173.967,25.804,154.545
C03191=1075.015,180.101,-76.485,173.970,25.807,154.545
C03192=1075.020,180.350,-76.508,173.971,25.809,154.545
C03193=1075.026,180.600,-76.530,173.974,25.811,154.546
C03194=1075.032,180.848,-76.552,173.976,25.815,154.546
C03195=1075.037,181.096,-76.575,173.977,25.817,154.546
C03196=1075.043,181.345,-76.598,173.980,25.819,154.547
C03197=1075.048,181.595,-76.620,173.982,25.822,154.547
C03198=1075.055,181.843,-76.642,173.985,25.825,154.547
C03199=1075.061,182.092,-76.665,173.986,25.827,154.547
C03200=1075.066,182.341,-76.688,173.988,25.830,154.548
C03201=1075.072,182.590,-76.711,173.991,25.833,154.548
C03202=1075.078,182.840,-76.733,173.992,25.835,154.548
C03203=1075.084,183.088,-76.756,173.995,25.837,154.549
C03204=1075.090,183.337,-76.779,173.997,25.840,154.549
C03205=1075.095,183.586,-76.802,173.999,25.843,154.549
C03206=1075.101,183.835,-76.825,174.001,25.845,154.549
C03207=1075.107,184.084,-76.848,174.003,25.848,154.550
C03208=1075.113,184.332,-76.870,174.006,25.851,154.550
C03209=1075.119,184.581,-76.893,174.007,25.853,154.550
C03210=1075.125,184.831,-76.915,174.009,25.856,154.551
C03211=1075.130,185.080,-76.938,174.012,25.858,154.551
C03212=1075.135,185.328,-76.961,174.014,25.861,154.551
C03213=1075.140,185.577,-76.984,174.016,25.863,154.552
C03214=1075.146,185.826,-77.007,174.018,25.867,154.552
C03215=1075.152,186.075,-77.030,174.020,25.869,154.552
C03216=1075.158,186.324,-77.053,174.023,25.872,154.552
C03217=1075.163,186.573,-77.076,174.024,25.875,154.553
C03218=1075.168,186.822,-77.099,174.027,25.877,154.553
C03219=1075.174,187.071,-77.122,174.029,25.880,154.553
C03220=1075.180,187.320,-77.145,174.031,25.883,154.554
C03221=1075.185,187.568,-77.168,174.033,25.885,154.554
C03222=1075.190,187.817,-77.191,174.035,25.888,154.554
C03223=1075.196,188.066,-77.214,174.037,25.891,154.555
C03224=1075.202,188.314,-77.238,174.040,25.893,154.555
C03225=1075.207,188.563,-77.261,174.041,25.896,154.555
C03226=1075.212,188.812,-77.285,174.044,25.899,154.556
C03227=1075.218,189.061,-77.307,174.046,25.902,154.556
C03228=1075.224,189.310,-77.330,174.048,25.905,154.556
C03229=1075.230,189.559,-77.353,174.050,25.907,154.557
C03230=1075.235,189.808,-77.377,174.052,25.910,154.557
C03231=1075.240,190.057,-77.400,174.054,25.913,154.557
C03232=1075.246,190.305,-77.424,174.057,25.915,154.558
C03233=1075.251,190.555,-77.447,174.058,25.918,154.558
C03234=1075.257,190.804,-77.470,174.061,25.920,154.558
C03235=1075.263,191.084,-77.495,174.063,25.924,154.559
C03236=1075.269,191.365,-77.522,174.065,25.927,154.559
C03237=1075.276,191.647,-77.549,174.069,25.930,154.559
C03238=1075.283,191.927,-77.575,174.071,25.933,154.560
C03239=1075.288,192.176,-77.598,174.073,25.936,154.560
C03240=1075.293,192.425,-77.621,174.075,25.938,154.560
C03241=1075.299,192.673,-77.645,174.077,25.941,154.561
C03242=1075.304,192.922,-77.668,174.079,25.944,154.561
C03243=1075.310,193.171,-77.691,174.082,25.946,154.561
C03244=1075.316,193.420,-77.714,174.084,25.949,154.561
C03245=1075.321,193.669,-77.738,174.086,25.952,154.562
C03246=1075.327,193.918,-77.761,174.088,25.954,154.562
C03247=1075.333,194.166,-77.784,174.090,25.957,154.562
C03248=1075.338,194.415,-77.809,174.093,25.960,154.563
C03249=1075.344,194.664,-77.832,174.095,25.963,154.563
C03250=1075.350,194.914,-77.855,174.097,25.965,154.563
C03251=1075.355,195.162,-77.879,174.099,25.968,154.564
C03252=1075.361,195.411,-77.902,174.101,25.971,154.564
C03253=1075.367,195.659,-77.926,174.104,25.973,154.564
C03254=1075.372,195.908,-77.949,174.106,25.976,154.565
C03255=1075.378,196.157,-77.972,174.107,25.979,154.565
C03256=1075.384,196.406,-77.996,174.110,25.981,154.565
C03257=1075.389,196.655,-78.019,174.112,25.984,154.566
C03258=1075.395,196.903,-78.043,174.115,25.987,154.566
C03259=1075.401,197.153,-78.066,174.117,25.989,154.566
C03260=1075.406,197.401,-78.091,174.119,25.992,154.567
C03261=1075.412,197.650,-78.114,174.121,25.995,154.567
C03262=1075.417,197.899,-78.138,174.123,25.997,154.567
C03263=1075.423,198.148,-78.161,174.125,26.000,154.567
C03264=1075.429,198.396,-78.184,174.128,26.003,154.568
C03265=1075.435,198.646,-78.208,174.130,26.006,154.568
C03266=1075.441,198.894,-78.232,174.133,26.009,154.568
C03267=1075.446,199.143,-78.256,174.135,26.011,154.569
C03268=1075.452,199.392,-78.279,174.137,26.013,154.569
C03269=1075.458,199.641,-78.302,174.139,26.017,154.569
C03270=1075.463,199.890,-78.327,174.141,26.019,154.570
C03271=1075.469,200.138,-78.350,174.144,26.022,154.570
C03272=1075.474,200.387,-78.374,174.146,26.025,154.570
C03273=1075.481,200.636,-78.398,174.148,26.027,154.571
C03274=1075.486,200.884,-78.421,174.151,26.030,154.571
C03275=1075.492,201.134,-78.445,174.152,26.033,154.571
C03276=1075.498,201.382,-78.469,174.155,26.035,154.571
C03277=1075.503,201.631,-78.492,174.157,26.038,154.572
C03278=1075.509,201.880,-78.516,174.159,26.040,154.572
C03279=1075.515,202.129,-78.541,174.162,26.044,154.572
C03280=1075.521,202.378,-78.564,174.164,26.046,154.573
C03281=1075.526,202.626,-78.588,174.167,26.049,154.573
C03282=1075.532,202.875,-78.612,174.169,26.052,154.573
C03283=1075.538,203.124,-78.636,174.171,26.054,154.574
C03284=1075.543,203.373,-78.660,174.173,26.057,154.574
C03285=1075.549,203.621,-78.683,174.175,26.060,154.574
C03286=1075.554,203.870,-78.708,174.177,26.063,154.575
C03287=1075.560,204.119,-78.732,174.180,26.065,154.575
C03288=1075.566,204.368,-78.755,174.182,26.069,154.575
C03289=1075.571,204.617,-78.780,174.185,26.071,154.576
C03290=1075.577,204.865,-78.804,174.187,26.074,154.576
C03291=1075.582,205.114,-78.828,174.189,26.077,154.576
C03292=1075.589,205.363,-78.852,174.192,26.080,154.577
C03293=1075.594,205.611,-78.876,174.193,26.082,154.577
C03294=1075.599,205.861,-78.900,174.196,26.085,154.577
C03295=1075.605,206.109,-78.923,174.198,26.088,154.578
C03296=1075.611,206.358,-78.948,174.200,26.090,154.578
C03297=1075.616,206.607,-78.972,174.203,26.093,154.578
C03298=1075.621,206.855,-78.997,174.205,26.096,154.578
C03299=1075.645,207.893,-79.097,174.322,26.158,154.579
C03300=1075.655,208.304,-79.139,174.325,26.164,154.579
C03301=1075.665,208.714,-79.179,174.329,26.170,154.580
C03302=1075.675,209.125,-79.220,174.332,26.176,154.581
C03303=1075.684,209.535,-79.261,174.336,26.182,154.582
C03304=1075.690,209.784,-79.285,174.338,26.186,154.583
C03305=1075.696,210.032,-79.311,174.340,26.190,154.583
C03306=1075.701,210.281,-79.335,174.342,26.194,154.584
C03307=1075.707,210.530,-79.360,174.345,26.197,154.584
C03308=1075.712,210.779,-79.385,174.347,26.201,154.585
C03309=1075.718,211.027,-79.410,174.349,26.205,154.585
C03310=1075.724,211.277,-79.435,174.351,26.209,154.586
C03311=1075.730,211.525,-79.460,174.353,26.212,154.586
C03312=1075.736,211.773,-79.485,174.356,26.216,154.587
C03313=1075.741,212.022,-79.510,174.358,26.220,154.588
C03314=1075.747,212.270,-79.535,174.360,26.224,154.588
C03315=1075.753,212.520,-79.560,174.362,26.227,154.589
C03316=1075.758,212.768,-79.585,174.364,26.231,154.589
C03317=1075.764,213.017,-79.611,174.366,26.235,154.590
C03318=1075.770,213.266,-79.635,174.369,26.238,154.590
C03319=1075.776,213.514,-79.660,174.371,26.242,154.591
C03320=1075.782,213.763,-79.685,174.373,26.246,154.591
C03321=1075.786,214.012,-79.710,174.375,26.250,154.592
C03322=1075.793,214.260,-79.736,174.377,26.253,154.592
C03323=1075.799,214.509,-79.761,174.379,26.257,154.593
C03324=1075.804,214.757,-79.785,174.382,26.261,154.594
C03325=1075.810,215.006,-79.811,174.384,26.265,154.594
C03326=1075.816,215.255,-79.837,174.386,26.268,154.595
C03327=1075.821,215.503,-79.862,174.388,26.272,154.595
C03328=1075.827,215.753,-79.887,174.390,26.276,154.596
C03329=1075.833,216.001,-79.912,174.392,26.280,154.596
C03330=1075.838,216.249,-79.937,174.395,26.283,154.597
C03331=1075.844,216.498,-79.963,174.397,26.287,154.597
C03332=1075.850,216.747,-79.988,174.399,26.290,154.598
C03333=1075.856,216.995,-80.013,174.401,26.295,154.599
C03334=1075.862,217.244,-80.038,174.403,26.298,154.599
C03335=1075.867,217.493,-80.064,174.406,26.302,154.600
C03336=1075.873,217.742,-80.089,174.408,26.305,154.600
C03337=1075.879,217.990,-80.114,174.410,26.309,154.601
C03338=1075.884,218.239,-80.140,174.412,26.313,154.601
C03339=1075.891,218.487,-80.165,174.414,26.317,154.602
C03340=1075.897,218.736,-80.191,174.417,26.320,154.602
C03341=1075.902,218.984,-80.216,174.419,26.324,154.603
C03342=1075.908,219.233,-80.242,174.421,26.328,154.603
C03343=1075.914,219.482,-80.267,174.423,26.331,154.604
C03344=1075.919,219.731,-80.292,174.425,26.335,154.604
C03345=1075.925,219.980,-80.318,174.427,26.339,154.605
C03346=1075.930,220.228,-80.343,174.430,26.342,154.606
C03347=1075.937,220.477,-80.368,174.432,26.346,154.606
C03348=1075.943,220.726,-80.394,174.434,26.350,154.607
C03349=1075.948,220.974,-80.420,174.436,26.353,154.607
C03350=1075.955,221.223,-80.446,174.439,26.357,154.608
C03351=1075.960,221.471,-80.471,174.441,26.360,154.608
C03352=1075.970,221.886,-80.514,174.445,26.367,154.609
C03353=1075.979,222.300,-80.556,174.449,26.374,154.610
C03354=1075.989,222.715,-80.599,174.453,26.379,154.611
C03355=1075.998,223.130,-80.642,174.456,26.386,154.612
C03356=1076.004,223.378,-80.667,174.458,26.389,154.612
C03357=1076.010,223.627,-80.694,174.461,26.393,154.613
C03358=1076.015,223.876,-80.720,174.463,26.397,154.613
C03359=1076.021,224.124,-80.745,174.465,26.401,154.614
C03360=1076.026,224.373,-80.771,174.467,26.404,154.614
C03361=1076.032,224.621,-80.796,174.469,26.408,154.615
C03362=1076.038,224.870,-80.823,174.472,26.412,154.616
C03363=1076.044,225.119,-80.849,174.474,26.416,154.616
C03364=1076.050,225.367,-80.874,174.476,26.419,154.617
C03365=1076.055,225.616,-80.900,174.478,26.423,154.617
C03366=1076.062,225.864,-80.926,174.481,26.427,154.618
C03367=1076.067,226.113,-80.952,174.484,26.430,154.618
C03368=1076.072,226.362,-80.978,174.486,26.434,154.619
C03369=1076.078,226.610,-81.003,174.488,26.438,154.619
C03370=1076.084,226.859,-81.030,174.490,26.442,154.620
C03371=1076.090,227.108,-81.055,174.492,26.445,154.620
C03372=1076.096,227.356,-81.081,174.495,26.449,154.621
C03373=1076.102,227.605,-81.107,174.497,26.452,154.621
C03374=1076.107,227.854,-81.133,174.499,26.456,154.622
C03375=1076.114,228.102,-81.159,174.501,26.460,154.623
C03376=1076.119,228.351,-81.185,174.503,26.464,154.623
C03377=1076.125,228.600,-81.211,174.506,26.467,154.624
C03378=1076.131,228.848,-81.237,174.509,26.471,154.624
C03379=1076.137,229.097,-81.263,174.511,26.475,154.625
C03380=1076.142,229.345,-81.290,174.513,26.478,154.625
C03381=1076.149,229.594,-81.315,174.515,26.482,154.626
C03382=1076.154,229.842,-81.342,174.518,26.485,154.626
C03383=1076.160,230.091,-81.368,174.520,26.490,154.627
C03384=1076.166,230.339,-81.394,174.522,26.493,154.627
C03385=1076.172,230.588,-81.420,174.524,26.497,154.628
C03386=1076.178,230.836,-81.446,174.527,26.500,154.628
C03387=1076.183,231.085,-81.472,174.530,26.504,154.629
C03388=1076.189,231.334,-81.499,174.532,26.508,154.630
C03389=1076.194,231.583,-81.525,174.534,26.512,154.630
C03390=1076.200,231.831,-81.552,174.536,26.516,154.631
C03391=1076.206,232.079,-81.578,174.539,26.519,154.631
C03392=1076.212,232.328,-81.604,174.541,26.523,154.632
C03393=1076.218,232.576,-81.630,174.543,26.526,154.632
C03394=1076.223,232.825,-81.656,174.545,26.530,154.633
C03395=1076.229,233.074,-81.683,174.547,26.534,154.633
C03396=1076.235,233.322,-81.709,174.551,26.538,154.634
C03397=1076.240,233.571,-81.735,174.553,26.541,154.634
C03398=1076.246,233.820,-81.762,174.555,26.545,154.635
C03399=1076.252,234.068,-81.789,174.557,26.549,154.635
C03400=1076.258,234.316,-81.815,174.559,26.553,154.636
C03401=1076.263,234.565,-81.841,174.562,26.556,154.637
C03402=1076.269,234.814,-81.868,174.564,26.560,154.637
C03403=1076.275,235.062,-81.895,174.566,26.563,154.638
C03404=1076.284,235.468,-81.938,174.571,26.570,154.639
C03405=1076.293,235.874,-81.981,174.574,26.576,154.639
C03406=1076.303,236.281,-82.024,174.578,26.582,154.640
C03407=1076.313,236.687,-82.068,174.582,26.588,154.641
C03408=1076.318,236.935,-82.095,174.584,26.592,154.642
C03409=1076.324,237.184,-82.121,174.586,26.596,154.642
C03410=1076.329,237.433,-82.148,174.588,26.599,154.643
C03411=1076.335,237.681,-82.174,174.592,26.603,154.643
C03412=1076.341,237.930,-82.201,174.594,26.607,154.644
C03413=1076.346,238.178,-82.228,174.596,26.610,154.644
C03414=1076.352,238.426,-82.254,174.598,26.614,154.645
C03415=1076.358,238.675,-82.281,174.601,26.617,154.645
C03416=1076.364,238.924,-82.308,174.603,26.621,154.646
C03417=1076.370,239.172,-82.335,174.606,26.625,154.647
C03418=1076.376,239.421,-82.361,174.608,26.629,154.647
C03419=1076.382,239.669,-82.388,174.610,26.632,154.648
C03420=1076.387,239.917,-82.415,174.613,26.636,154.648
C03421=1076.394,240.166,-82.442,174.615,26.640,154.649
C03422=1076.399,240.415,-82.469,174.617,26.644,154.649
C03423=1076.404,240.663,-82.495,174.620,26.648,154.650
C03424=1076.410,240.912,-82.522,174.623,26.651,154.650
C03425=1076.416,241.160,-82.549,174.625,26.655,154.651
C03426=1076.422,241.409,-82.576,174.627,26.658,154.651
C03427=1076.428,241.658,-82.602,174.629,26.662,154.652
C03428=1076.434,241.906,-82.629,174.632,26.665,154.652
C03429=1076.439,242.155,-82.656,174.635,26.669,154.653
C03430=1076.445,242.402,-82.684,174.637,26.673,154.654
C03431=1076.451,242.651,-82.711,174.639,26.677,154.654
C03432=1076.457,242.900,-82.737,174.641,26.681,154.655
C03433=1076.462,243.148,-82.765,174.644,26.684,154.655
C03434=1076.468,243.397,-82.791,174.647,26.688,154.656
C03435=1076.474,243.645,-82.818,174.649,26.692,154.656
C03436=1076.480,243.894,-82.846,174.651,26.696,154.657
C03437=1076.486,244.142,-82.873,174.653,26.699,154.657
C03438=1076.491,244.391,-82.899,174.656,26.703,154.658
C03439=1076.496,244.639,-82.927,174.659,26.707,154.658
C03440=1076.503,244.888,-82.954,174.661,26.711,154.659
C03441=1076.509,245.136,-82.981,174.663,26.714,154.660
C03442=1076.514,245.385,-83.008,174.666,26.718,154.660
C03443=1076.520,245.632,-83.036,174.668,26.721,154.661
C03444=1076.526,245.882,-83.063,174.671,26.726,154.661
C03445=1076.531,246.130,-83.090,174.673,26.729,154.662
C03446=1076.537,246.378,-83.117,174.675,26.733,154.662
C03447=1076.542,246.627,-83.145,174.678,26.736,154.663
C03448=1076.549,246.876,-83.172,174.680,26.740,154.663
C03449=1076.554,247.124,-83.200,174.683,26.744,154.664
C03450=1076.560,247.372,-83.226,174.685,26.748,154.664
C03451=1076.566,247.621,-83.254,174.688,26.752,154.665
C03452=1076.572,247.869,-83.281,174.690,26.755,154.666
C03453=1076.577,248.118,-83.308,174.693,26.759,154.666
C03454=1076.583,248.366,-83.336,174.695,26.763,154.667
C03455=1076.588,248.615,-83.363,174.697,26.767,154.667
C03456=1076.597,249.014,-83.408,174.701,26.773,154.668
C03457=1076.607,249.414,-83.452,174.705,26.779,154.669
C03458=1076.616,249.814,-83.496,174.710,26.785,154.670
C03459=1076.625,250.213,-83.540,174.713,26.791,154.671
C03460=1076.631,250.461,-83.568,174.716,26.795,154.671
C03461=1076.636,250.710,-83.595,174.718,26.799,154.672
C03462=1076.642,250.958,-83.623,174.721,26.802,154.672
C03463=1076.648,251.206,-83.651,174.723,26.806,154.673
C03464=1076.653,251.455,-83.678,174.725,26.810,154.674
C03465=1076.659,251.703,-83.706,174.728,26.814,154.674
C03466=1076.665,251.952,-83.733,174.731,26.817,154.675
C03467=1076.670,252.200,-83.761,174.733,26.821,154.675
C03468=1076.676,252.448,-83.789,174.735,26.825,154.676
C03469=1076.683,252.697,-83.817,174.738,26.829,154.676
C03470=1076.688,252.946,-83.844,174.741,26.832,154.677
C03471=1076.693,253.194,-83.872,174.743,26.836,154.677
C03472=1076.700,253.442,-83.900,174.745,26.840,154.678
C03473=1076.705,253.691,-83.927,174.748,26.844,154.679
C03474=1076.711,253.940,-83.955,174.751,26.847,154.679
C03475=1076.717,254.187,-83.983,174.753,26.851,154.680
C03476=1076.723,254.436,-84.011,174.755,26.855,154.680
C03477=1076.728,254.684,-84.039,174.757,26.859,154.681
C03478=1076.734,254.932,-84.066,174.761,26.862,154.681
C03479=1076.740,255.181,-84.094,174.763,26.866,154.682
C03480=1076.745,255.429,-84.122,174.765,26.870,154.682
C03481=1076.752,255.678,-84.150,174.768,26.874,154.683
C03482=1076.757,255.926,-84.178,174.771,26.877,154.683
C03483=1076.763,256.174,-84.206,174.773,26.881,154.684
C03484=1076.768,256.423,-84.234,174.775,26.885,154.685
C03485=1076.775,256.672,-84.261,174.778,26.889,154.685
C03486=1076.780,256.920,-84.289,174.781,26.892,154.686
C03487=1076.786,257.168,-84.317,174.783,26.896,154.686
C03488=1076.791,257.416,-84.345,174.786,26.900,154.687
C03489=1076.798,257.665,-84.373,174.788,26.903,154.687
C03490=1076.803,257.913,-84.401,174.790,26.907,154.688
C03491=1076.809,258.162,-84.429,174.793,26.911,154.688
C03492=1076.815,258.410,-84.457,174.796,26.915,154.689
C03493=1076.821,258.658,-84.485,174.798,26.918,154.689
C03494=1076.827,258.907,-84.513,174.801,26.922,154.690
C03495=1076.833,259.155,-84.541,174.804,26.926,154.691
C03496=1076.839,259.404,-84.569,174.806,26.930,154.691
C03497=1076.845,259.651,-84.597,174.808,26.933,154.692
C03498=1076.851,259.900,-84.625,174.811,26.937,154.692
C03499=1076.857,260.148,-84.654,174.814,26.941,154.693
C03500=1076.862,260.396,-84.682,174.816,26.944,154.693
C03501=1076.868,260.645,-84.710,174.819,26.949,154.694
C03502=1076.875,260.894,-84.738,174.821,26.952,154.694
C03503=1076.880,261.142,-84.766,174.824,26.956,154.695
C03504=1076.886,261.390,-84.794,174.827,26.960,154.695
C03505=1076.891,261.638,-84.822,174.829,26.963,154.696
C03506=1076.898,261.887,-84.851,174.832,26.967,154.696
C03507=1076.904,262.135,-84.879,174.835,26.971,154.697
C03508=1076.913,262.532,-84.925,174.838,26.977,154.698
C03509=1076.922,262.929,-84.970,174.842,26.982,154.699
C03510=1076.932,263.326,-85.015,174.847,26.988,154.700
C03511=1076.942,263.723,-85.060,174.851,26.994,154.700
C03512=1076.948,263.971,-85.089,174.853,26.998,154.701
C03513=1076.953,264.219,-85.117,174.856,27.002,154.702
C03514=1076.960,264.467,-85.146,174.859,27.005,154.702
C03515=1076.966,264.716,-85.174,174.861,27.010,154.703
C03516=1076.971,264.964,-85.202,174.864,27.013,154.703
C03517=1076.976,265.213,-85.232,174.866,27.017,154.704
C03518=1076.982,265.461,-85.260,174.869,27.021,154.704
C03519=1076.988,265.709,-85.289,174.872,27.025,154.705
C03520=1076.994,265.958,-85.317,174.874,27.028,154.705
C03521=1077.000,266.206,-85.345,174.876,27.032,154.706
C03522=1077.006,266.454,-85.374,174.880,27.036,154.707
C03523=1077.012,266.703,-85.402,174.882,27.040,154.707
C03524=1077.018,266.951,-85.431,174.884,27.044,154.708
C03525=1077.022,267.199,-85.460,174.887,27.048,154.708
C03526=1077.029,267.447,-85.489,174.890,27.051,154.709
C03527=1077.035,267.696,-85.517,174.892,27.055,154.709
C03528=1077.041,267.944,-85.546,174.895,27.059,154.710
C03529=1077.046,268.192,-85.574,174.897,27.062,154.710
C03530=1077.052,268.440,-85.603,174.901,27.066,154.711
C03531=1077.058,268.689,-85.633,174.903,27.070,154.712
C03532=1077.064,268.937,-85.661,174.905,27.074,154.712
C03533=1077.070,269.185,-85.690,174.908,27.078,154.713
C03534=1077.075,269.434,-85.718,174.910,27.082,154.713
C03535=1077.082,269.682,-85.747,174.913,27.085,154.714
C03536=1077.087,269.930,-85.777,174.916,27.089,154.714
C03537=1077.093,270.178,-85.805,174.918,27.093,154.715
C03538=1077.099,270.426,-85.834,174.921,27.097,154.716
C03539=1077.104,270.675,-85.863,174.924,27.100,154.716
C03540=1077.111,270.923,-85.892,174.926,27.104,154.717
C03541=1077.117,271.172,-85.921,174.929,27.108,154.717
C03542=1077.122,271.419,-85.949,174.931,27.112,154.718
C03543=1077.128,271.668,-85.979,174.935,27.116,154.718
C03544=1077.134,271.916,-86.008,174.937,27.120,154.719
C03545=1077.140,272.165,-86.036,174.939,27.124,154.720
C03546=1077.145,272.413,-86.066,174.942,27.127,154.720
C03547=1077.151,272.660,-86.095,174.945,27.131,154.721
C03548=1077.157,272.909,-86.124,174.948,27.135,154.721
C03549=1077.163,273.157,-86.153,174.950,27.139,154.722
C03550=1077.169,273.406,-86.182,174.952,27.142,154.722
C03551=1077.174,273.654,-86.211,174.956,27.147,154.723
C03552=1077.180,273.902,-86.240,174.958,27.150,154.723
C03553=1077.185,274.150,-86.270,174.961,27.154,154.724
C03554=1077.192,274.398,-86.299,174.963,27.158,154.725
C03555=1077.198,274.646,-86.328,174.966,27.162,154.725
C03556=1077.203,274.895,-86.357,174.969,27.166,154.726
C03557=1077.210,275.143,-86.386,174.971,27.169,154.726
C03558=1077.215,275.391,-86.416,174.974,27.174,154.727
C03559=1077.221,275.639,-86.445,174.977,27.177,154.727
C03560=1077.230,276.040,-86.492,174.981,27.184,154.728
C03561=1077.240,276.439,-86.539,174.985,27.190,154.729
C03562=1077.249,276.840,-86.587,174.990,27.196,154.730
C03563=1077.259,277.239,-86.634,174.994,27.202,154.731
C03564=1077.264,277.487,-86.664,174.997,27.206,154.732
C03565=1077.270,277.736,-86.693,174.999,27.210,154.732
C03566=1077.276,277.984,-86.722,175.002,27.214,154.733
C03567=1077.281,278.232,-86.752,175.005,27.218,154.733
C03568=1077.288,278.481,-86.781,175.008,27.222,154.734
C03569=1077.293,278.729,-86.811,175.010,27.225,154.735
C03570=1077.299,278.977,-86.840,175.012,27.229,154.735
C03571=1077.305,279.225,-86.870,175.016,27.233,154.736
C03572=1077.311,279.473,-86.900,175.018,27.237,154.736
C03573=1077.317,279.721,-86.929,175.021,27.241,154.737
C03574=1077.322,279.970,-86.959,175.023,27.245,154.738
C03575=1077.329,280.217,-86.988,175.027,27.249,154.738
C03576=1077.335,280.466,-87.018,175.029,27.252,154.739
C03577=1077.340,280.714,-87.048,175.032,27.257,154.739
C03578=1077.346,280.962,-87.077,175.034,27.260,154.740
C03579=1077.352,281.210,-87.107,175.038,27.264,154.740
C03580=1077.358,281.459,-87.137,175.040,27.268,154.741
C03581=1077.363,281.707,-87.166,175.042,27.272,154.742
C03582=1077.369,281.955,-87.197,175.045,27.276,154.742
C03583=1077.375,282.203,-87.226,175.048,27.280,154.743
C03584=1077.381,282.451,-87.256,175.051,27.284,154.743
C03585=1077.387,282.699,-87.286,175.053,27.288,154.744
C03586=1077.392,282.948,-87.315,175.056,27.292,154.745
C03587=1077.398,283.196,-87.346,175.059,27.296,154.745
C03588=1077.404,283.444,-87.375,175.062,27.300,154.746
C03589=1077.410,283.692,-87.405,175.064,27.304,154.746
C03590=1077.415,283.940,-87.435,175.067,27.307,154.747
C03591=1077.421,284.188,-87.465,175.070,27.311,154.748
C03592=1077.427,284.436,-87.495,175.073,27.315,154.748
C03593=1077.433,284.684,-87.524,175.075,27.319,154.749
C03594=1077.439,284.932,-87.554,175.078,27.324,154.749
C03595=1077.445,285.180,-87.584,175.081,27.327,154.750
C03596=1077.450,285.429,-87.614,175.084,27.331,154.751
C03597=1077.456,285.676,-87.644,175.086,27.335,154.751
C03598=1077.462,285.925,-87.675,175.089,27.339,154.752
C03599=1077.468,286.173,-87.705,175.091,27.343,154.752
C03600=1077.474,286.421,-87.734,175.095,27.347,154.753
C03601=1077.480,286.669,-87.765,175.097,27.351,154.754
C03602=1077.486,286.917,-87.794,175.100,27.355,154.754
C03603=1077.492,287.165,-87.825,175.103,27.359,154.755
C03604=1077.497,287.413,-87.855,175.106,27.362,154.755
C03605=1077.503,287.661,-87.885,175.108,27.366,154.756
C03606=1077.509,287.910,-87.915,175.111,27.371,154.757
C03607=1077.515,288.158,-87.946,175.114,27.374,154.757
C03608=1077.521,288.406,-87.975,175.117,27.379,154.758
C03609=1077.527,288.653,-88.005,175.120,27.382,154.758
C03610=1077.533,288.901,-88.036,175.122,27.386,154.759
C03611=1077.539,289.150,-88.066,175.125,27.391,154.760
C03612=1077.548,289.559,-88.116,175.129,27.397,154.761
C03613=1077.558,289.969,-88.166,175.134,27.403,154.761
C03614=1077.567,290.380,-88.216,175.139,27.410,154.763
C03615=1077.577,290.789,-88.267,175.143,27.417,154.763
C03616=1077.584,291.038,-88.297,175.147,27.421,154.764
C03617=1077.589,291.286,-88.328,175.149,27.425,154.765
C03618=1077.595,291.534,-88.358,175.152,27.429,154.765
C03619=1077.601,291.781,-88.388,175.154,27.433,154.766
C03620=1077.607,292.029,-88.419,175.158,27.437,154.767
C03621=1077.612,292.278,-88.450,175.160,27.441,154.767
C03622=1077.618,292.526,-88.480,175.163,27.445,154.768
C03623=1077.624,292.774,-88.511,175.165,27.449,154.768
C03624=1077.630,293.022,-88.541,175.169,27.453,154.769
C03625=1077.636,293.270,-88.572,175.172,27.457,154.770
C03626=1077.642,293.518,-88.602,175.174,27.461,154.770
C03627=1077.647,293.766,-88.633,175.177,27.465,154.771
C03628=1077.653,294.014,-88.663,175.180,27.469,154.772
C03629=1077.659,294.262,-88.694,175.183,27.473,154.772
C03630=1077.665,294.510,-88.724,175.185,27.477,154.773
C03631=1077.671,294.758,-88.755,175.188,27.481,154.773
C03632=1077.678,295.006,-88.786,175.192,27.485,154.774
C03633=1077.683,295.254,-88.817,175.194,27.489,154.775
C03634=1077.689,295.502,-88.848,175.197,27.493,154.775
C03635=1077.695,295.750,-88.878,175.199,27.497,154.776
C03636=1077.701,295.998,-88.909,175.203,27.501,154.776
C03637=1077.706,296.246,-88.940,175.206,27.506,154.777
C03638=1077.713,296.494,-88.971,175.208,27.509,154.778
C03639=1077.719,296.742,-89.001,175.211,27.514,154.778
C03640=1077.724,296.990,-89.032,175.214,27.517,154.779
